	// Set the mode
	IF ctrl.nLS_Mode <> E_CRYO_LAKESHORE_MODE.MONITORING THEN
		Lakeshore.M_SetMode(ctrl.nLS_Mode);
	ELSE
		RETURN;	// Nothing to do
	END_IF
ELSE
	RETURN;	// Nothing to do
END_IF




CASE ctrl.nLS_Mode OF
	E_CRYO_LAKESHORE_MODE.MONITORING,
	E_CRYO_LAKESHORE_MODE.COOLING,
	E_CRYO_LAKESHORE_MODE.WARMUP,
	E_CRYO_LAKESHORE_MODE.COOLING_UPDATE,
	E_CRYO_LAKESHORE_MODE.WARMUP_UPDATE:
		Lakeshore.M_SetMode(E_CRYO_LAKESHORE_MODE.MONITORING);	// No action
		
	E_CRYO_LAKESHORE_MODE.SINGLE_SETUP:
		IF stat.nState = E_CRYO_CTRL_STATE.COLD THEN
			Lakeshore.M_SetParams(
				in_nPID_A_P			:= cfg.LS_W_PID_A_P, 
				in_nPID_A_I			:= cfg.LS_W_PID_A_I, 
				in_nPID_A_D			:= cfg.LS_W_PID_A_D, 
				in_nHeater_Range	:= cfg.LS_W_Heater_Range, 
				in_lrCtrlRamp		:= ctrl.lrLS_RAMP, 
				in_lrSetpoint_A		:= ctrl.lrLS_SETP);
		END_IF
	ELSE
		Lakeshore.M_SetMode(E_CRYO_LAKESHORE_MODE.MONITORING);	// No action
END_CASE
*)
END_METHOD

// Method to check status of the cryostat vacuum.
// TODO: The limits might depend on the temperature.
METHOD M_CheckVacuum
VAR_INPUT
END_VAR
//IF Pressure_Cryo.stat.bValid  THEN
//	IF Pressure_Cryo.stat.lrPressure < cfg.lrPress_GoodVac THEN
//		stat.bInVacuum	:= TRUE;
//		stat.bGoodVacuum:= TRUE;
//	ELSIF Pressure_Cryo.stat.lrPressure < cfg.lrPress_InVac THEN
//		stat.bInVacuum	:= TRUE;
//		stat.bGoodVacuum:= FALSE;
//	ELSE
//		stat.bInVacuum	:= FALSE;
//		stat.bGoodVacuum:= FALSE;
//	END_IF 
//ELSE
//	stat.bInVacuum	:= FALSE;
//	stat.bGoodVacuum:= FALSE;
//END_IF
END_METHOD

METHOD M_Configure
VAR_INPUT
END_VAR

IF NOT stat.bConfigured THEN
	

// This call just configures logs at the very start.
// Logging is done by explicit calls to M_LogInfo().
logs(in_sName := in_sName);

bPwr_VAG_PTA := TRUE;
bPwr_VAG_PTB := TRUE;
bPwr_VAG_PTC := TRUE;

	////////////////////
	// Coolant Valves//
	//////////////////
// Set pointers to Valves - MUST!!!
	ptrV[1]	:= ADR(TPC_A);
	ptrV[2]	:= ADR(TPC_B);
	
	
	// Set pointers to Valve Commands - MUST!!!
	ptrVC[1]	:= ADR(ctrl.cor_TPC_A);
	ptrVC[2]	:= ADR(ctrl.cor_TPC_B);
	
	
	// Set pointers to Enable Valves flags - MUST!!!
	ptrEV[1]	:= ADR(ctrl.bEnable_TPC_A);
	ptrEV[2]	:= ADR(ctrl.bEnable_TPC_B);









stat.bConfigured := TRUE;

END_IF 















//IF stat.bConfigured THEN
//	RETURN;
//ELSIF stat.nCycleCounter = 100 THEN
//	// Set pointers to system logs.
//	ptrLog[0] := ADR(syslog.s0);
//	ptrLog[1] := ADR(syslog.s1);
//	ptrLog[2] := ADR(syslog.s2);
//	ptrLog[3] := ADR(syslog.s3);
//	ptrLog[4] := ADR(syslog.s4);
//	ptrLog[5] := ADR(syslog.s5);
//	ptrLog[6] := ADR(syslog.s6);
//	ptrLog[7] := ADR(syslog.s7);
//	ptrLog[8] := ADR(syslog.s8);
//	ptrLog[9] := ADR(syslog.s9);
//ELSIF stat.nCycleCounter > 200 THEN
//	stat.bConfigured	:= TRUE;
//ELSE
//	RETURN;
//END_IF
END_METHOD

METHOD M_ExecuteControllers
VAR
END_VAR
VAR_INST
	trig_Turbo_ON:	R_TRIG;
	trig_Turbo_OFF:	F_TRIG;
END_VAR

met_tctrl(temperatures := met_temp);

met_heaters(tctrl := met_tctrl);

met_ccus();

// Evacuation is enabled, Check Venting valves and if they are open
// then Close them.
// Open PVV_P1 and Close PVV_P2 & PVV_P3
//IF met_evac.bEnable_met_evac THEN
//	IF met_venting.N2V_1.stat.bActON THEN
//		met_venting.in_bEnable_N2V_1 := FALSE;
//	END_IF
//	IF met_venting.N2V_2.stat.bActON THEN
//		met_venting.in_bEnable_N2V_2 := FALSE;
//	END_IF
	
//	met_cool_down.in_bEnable_PVV_P1:=	TRUE;
//	met_cool_down.in_bEnable_PVV_P2:=	FALSE;
//	met_cool_down.in_bEnable_PVV_P3:=	FALSE;
	
//	met_evac.stat.bInterlock := FALSE;
	
//END_IF


met_evac(in_Cryo_Stat := 						stat,
			interlocks:= 						interlocks);

//////////////////////////////////////////////
//             Venting
//////////////////////////////////////////////


met_venting(in_Cryo_Stat := 						stat,
			interlocks:= 						interlocks);

//////////////////////////////////////////////
//             Cool-Down
//////////////////////////////////////////////



met_cool_down(
	in_Cryo_Stat:=  							stat,
	in_lrLN2_TempK:= 							cfg.lrCoolDown_LN2_TempK,
	in_lrRadShld_TempK_TO_Start_PTCs:= 			cfg.lrRadShld_TempK_TO_Start_PTCs, 
	in_lrCoolDown_PreCond_Press:= 				cfg.lrCoolDown_PreCond_Press, 
	out_bCoolDownActive=> 						stat.bCoolDownActive, 
	all_cryo_temps:= 							met_temp, 
	all_heaters:= 								met_heaters, 
	all_t_ctrls:= 								met_tctrl, 
	all_t_votes:= 								met_voters, 
	interlocks:= 								interlocks);	





//////////////////////////////////////////////
//             Warmm_Up
//////////////////////////////////////////////

met_warm_up(
	in_Cryo_Stat:= 								stat, 
	in_lrWarmUp_Detectors_Ramp_1:= 				cfg.lrWarmUp_Detectors_Ramp_1, 
	in_lrWarmUp_Detectors_Ramp_Switch_Temp:=   	cfg.lrWarmUp_Detectors_Ramp_Switch_Temp, 
	in_lrWarmUp_Detectors_Ramp_2:=            	cfg.lrWarmUp_Detectors_Ramp_2,			
	in_lrWarmUp_EvacPermission_Temp:=         	cfg.lrWarmUp_EvacPermission_Temp,		
	in_lrWarmUp_VentingPermission_Temp:=      	cfg.lrWarmUp_VentingPermission_Temp,	
	in_lrWarmUp_Alarm_Temp:=                  	cfg.lrWarmUp_Alarm_Temp,				
	in_lrWarmUp_Alarm_PreCooling_Pressure:=   	cfg.lrWarmUp_Alarm_PreCooling_Pressure,
	out_bWarmUpActive=> 						stat.bWarmUpActive, 
	all_cryo_temps:= 							met_temp, 
	all_heaters:= 								met_heaters, 
	all_t_ctrls:= 								met_tctrl, 
	all_t_votes:= 								met_voters, 
	interlocks:= 								interlocks);



//////////////////////////////////////////////
//             Re_generation
//////////////////////////////////////////////


met_regeneration(
	in_Cryo_Stat:= 								stat, 
	in_lrRegeneration_Safe_Temp:= 				cfg.lrRegeneration_Safe_Temp, 
	in_lrRegeneration_Safe_Press:= 				cfg.lrRegeneration_Safe_Press, 
	in_lrTemp_Regeneration_SetPoint:= 			cfg.lrTemp_Regeneration_SetPoint, 
	in_lrTemp_Regeneration_Alarm:= 				cfg.lrTemp_Regeneration_Alarm_Temp, 
	in_lrTemp_Regeneration_Stop:= 				cfg.lrTemp_Regeneration_Stop, 
	in_tSorption_Pump_Cool_Down_TimeOut:= 		cfg.tSorption_Pump_Cool_Down_TimeOut, 
	out_bRegenerationActive=> 					stat.bRegenerationActive, 
	all_cryo_temps:= 							met_temp, 
	all_heaters:= 								met_heaters, 
	all_t_ctrls:= 								met_tctrl, 
	all_t_votes:=								met_voters, 
	interlocks:= 								interlocks);


//////////////////////////////////////////////
//             Anti-Fogging
//////////////////////////////////////////////


met_anti_fogging(
	//in_bEnable:= 								stat.bCoolDownActive, // Activate when Cool-down is active 
	in_Cryo_Stat:= 								stat, 
	in_lrAntiFog_Purging_DewPoint:= 			cfg.lrAntiFog_Purging_DewPoint, 
	in_lrAntiFog_Heating_DewPoint:= 			cfg.lrAntiFog_Heating_DewPoint, 
	in_lrAntiFog_DewPoint_Alarm:= 				cfg.lrAntiFog_DewPoint_Alarm, 
	out_bAntiFoggingActive=> 					stat.bAntiFoggingActive, 
	all_cryo_temps:= 							met_temp, 
	all_heaters:= 								met_heaters, 
	all_t_ctrls:= 								met_tctrl,   
	all_t_votes:=								met_voters,   
	interlocks:= 								interlocks);


//////////////////////////////////////////////
//             Coolant Valves
//////////////////////////////////////////////	

ctrl.cor_TPC_A(in_bEnable := ctrl.bEnable_TPC_A);	// Handling of PVV1 commands
ctrl.cor_TPC_B(in_bEnable := ctrl.bEnable_TPC_B);	// Handling of PVV2 commands

// Valve Control
TPC_A(
	in_bEnable			:= ctrl.cor_TPC_A.out_bEnable,
	in_nFeedback		:= E_CRYO_BIN_ACT_FEEDBACK.ON_ONLY);

TPC_B(
	in_bEnable			:= ctrl.cor_TPC_B.out_bEnable,
	in_nFeedback		:= E_CRYO_BIN_ACT_FEEDBACK.ON_ONLY);

// Reset valves

trig_Turbo_ON(CLK := stat.bTurboPumpsRunning);
trig_Turbo_OFF(CLK := stat.bTurboPumpsRunning);

IF trig_Turbo_ON.Q OR trig_Turbo_OFF.Q THEN
	TPC_A.M_Reset();
	TPC_B.M_Reset();
END_IF

// Actuate valves when turbo pumps are ON
ctrl.bEnable_TPC_A := stat.bTurboPumpsRunning;
ctrl.bEnable_TPC_B := stat.bTurboPumpsRunning;

	/////////////////////////////
	//// Time (NTP from ICS) /// 
	//////////////////////////

met_cry_time(in_diag_address:= , in_diag_destination_port:= , in_bDiagEnabled:= , in_nDefaultMode:= E_TIME_MODE.UTC_NTP);


	///////////////////////
	// xxxxxxxxxxxxxxxx //
	/////////////////////
	
	sim_regeneration();
END_METHOD

METHOD M_GetHighestTemperature
VAR_INPUT
END_VAR
VAR
	lrTempK:	LREAL	:= 0.0;	// The lowest possible temperature
	bValid:		BOOL	:= FALSE;
END_VAR
////
//// Get the warmest temperature among Mirror, Bench, FilterWheel and WarmUp
////

//// If there is at least one Valid reading, the result is valid.
//IF	Temp_Mirror.stat.bValid 	OR 
//	Temp_ColdBench.stat.bValid	OR 
//	Temp_FW.stat.bValid			OR 
//	Temp_WarmUp.stat.bValid			THEN
//	bValid	:= TRUE;
//END_IF


//// Get the highest temperature from Valid temperatures.
//// Take Mirror temperature first, if Valid.
//// If not Valid, try with WarmUp sensor.
//// If that doesn't work, take the Filter Wheel temperature.
//IF Temp_Mirror.stat.bValid THEN
//	IF Temp_Mirror.stat.lrTempK > lrTempK THEN
//		lrTempK	:= Temp_Mirror.stat.lrTempK;
//	END_IF
//ELSIF Temp_WarmUp.stat.bValid THEN
//	IF Temp_WarmUp.stat.lrTempK > lrTempK THEN
//		lrTempK	:= Temp_Mirror.stat.lrTempK;
//	END_IF
//ELSIF Temp_FW.stat.bValid THEN
//	IF Temp_FW.stat.lrTempK > lrTempK THEN
//		lrTempK	:= Temp_Mirror.stat.lrTempK;
//	END_IF
//END_IF


//// Update status
//stat.lrHighestTempK		:= lrTempK;
//stat.bHighestTempValid	:= bValid;
END_METHOD

METHOD M_GetLowestTemperature
VAR_INPUT
END_VAR
VAR
	lrTempK:	LREAL	:= 293.15;	// Room temperature 20 C
	bValid:		BOOL	:= FALSE;
END_VAR
////
//// Get the coldest temperature among Mirror, Bench, FilterWheel and WarmUp
////

//// If there is at least one Valid reading, the result is valid.
//IF	Temp_Mirror.stat.bValid 	OR 
//	Temp_ColdBench.stat.bValid	OR 
//	Temp_FW.stat.bValid			OR 
//	Temp_WarmUp.stat.bValid			THEN
//	bValid	:= TRUE;
//END_IF


//// Get the lowest temperature from Valid temperatures.
//IF Temp_Mirror.stat.bValid AND Temp_Mirror.stat.lrTempK < lrTempK THEN
//	lrTempK	:= Temp_Mirror.stat.lrTempK;
//END_IF

//IF Temp_ColdBench.stat.bValid AND Temp_ColdBench.stat.lrTempK < lrTempK THEN
//	lrTempK	:= Temp_ColdBench.stat.lrTempK;
//END_IF

//IF Temp_FW.stat.bValid AND Temp_FW.stat.lrTempK < lrTempK THEN
//	lrTempK	:= Temp_FW.stat.lrTempK;
//END_IF

//IF Temp_WarmUp.stat.bValid AND Temp_WarmUp.stat.lrTempK < lrTempK THEN
//	lrTempK	:= Temp_WarmUp.stat.lrTempK;
//END_IF

//// Update status
//stat.lrLowestTempK		:= lrTempK;
//stat.bLowestTempValid	:= bValid;

//// Get Temperature difference (DET -Lowest temperature) [K]
//IF stat.bLowestTempValid  AND  Temp_DET.stat.bValid  THEN
//	stat.bDiffTempValid	:= TRUE;
//	stat.lrDiffTempK	:= Temp_DET.stat.lrTempK - stat.lrLowestTempK;
//ELSE
//	stat.bDiffTempValid	:= FALSE;
//	stat.lrDiffTempK	:= -100;
//END_IF
END_METHOD

METHOD M_GetState
VAR_INPUT
END_VAR
VAR
	m_bIsCtrlOK           : BOOL;
    m_bIsWarm             : BOOL;
    m_bIsCold             : BOOL;
    m_bIsPartiallyCold    : BOOL;
    m_bIsInVacuum         : BOOL;
    m_bIsInPartialVacuum  : BOOL;
    m_bIsInGoodVacuum     : BOOL;
    m_bIsPressurized      : BOOL;

    m_nTmpState          : E_METIS_CRYO_CTRL_STATE;
    m_sStateDesc          : STRING;	

//    isCtrlOK: 			BOOL;
	
//    isWarm: 			BOOL;
//    isCold: 			BOOL;
//	isPartiallyCold: 	BOOL;
	
//    isInVacuum : 		BOOL;
//    isInPartialVacuum:	BOOL;
	
//	tempState : E_METIS_CRYO_CTRL_STATE;
END_VAR

m_bIsCtrlOK           := stat.bCtrlOK;
m_bIsWarm             := stat.bWarm;
m_bIsCold             := stat.bCold;
m_bIsPartiallyCold    := stat.bPartiallyCold;

m_bIsInVacuum         := stat.bInVacuum;
m_bIsInPartialVacuum  := stat.bPartialVacuum;
m_bIsInGoodVacuum     := stat.bInGoodVacuum;
m_bIsPressurized      := stat.bPressurized;


IF NOT m_bIsCtrlOK THEN
    m_nTmpState := E_METIS_CRYO_CTRL_STATE.ERROR;
    m_sStateDesc := 'Error: Controller is not OK';
	logs.M_LogInfo('');
	stat.bInitialized := FALSE;

ELSIF m_bIsWarm THEN
    IF m_bIsPressurized THEN
        m_nTmpState := E_METIS_CRYO_CTRL_STATE.WARM_PRESS;
        //m_sStateDesc := 'State: WarmPressurized';
		logs.M_LogInfo('System started in Warm-Pressurized state.');
		stat.bInitialized := TRUE;
    ELSIF m_bIsInVacuum THEN
        m_nTmpState := E_METIS_CRYO_CTRL_STATE.WARM_VACUUM;
        //m_sStateDesc := 'State: WarmVacuum';
		logs.M_LogInfo('System started in Warm-Vacuum state.');
		stat.bInitialized := TRUE;
    ELSIF m_bIsInPartialVacuum THEN
        m_nTmpState := E_METIS_CRYO_CTRL_STATE.PARTIAL_VACUUM;
        //m_sStateDesc := 'State: Partial Vacuum';
		logs.M_LogInfo('System started in Partial-Vacuum state');
		stat.bInitialized := TRUE;
    ELSE
        m_nTmpState := E_METIS_CRYO_CTRL_STATE.NONE;
        //m_sStateDesc := 'State Undefined: Warm with no pressure condition';
		logs.M_LogInfo('System started in undefined state: Warm with no pressure condition');
		stat.bInitialized := FALSE;
		ctrl.bEnable := FALSE;
    END_IF

ELSIF m_bIsCold THEN
	IF m_bIsInGoodVacuum THEN
    	m_nTmpState := E_METIS_CRYO_CTRL_STATE.COLD;
		logs.M_LogInfo('System started in Cold state');
		stat.bInitialized := TRUE;
	ELSE
		m_nTmpState := E_METIS_CRYO_CTRL_STATE.PARTIALLY_COLD;
		logs.M_LogInfo('System started in High Pressure & Low Temp state -> Start EVACUATION');
		stat.bInitialized := TRUE;
	END_IF

ELSIF m_bIsPartiallyCold THEN
    IF m_bIsInVacuum OR m_bIsInGoodVacuum THEN
        m_nTmpState := E_METIS_CRYO_CTRL_STATE.PARTIALLY_COLD;
       //m_sStateDesc := 'State: Partially Cold';
		logs.M_LogInfo('System started in Partially-Cold state.');
		stat.bInitialized := TRUE;
    ELSIF m_bIsPressurized THEN
        m_nTmpState := E_METIS_CRYO_CTRL_STATE.PARTIALLY_COLD;
        //m_sStateDesc := 'State: Partially Cold. Start EVACUATION';
		logs.M_LogInfo('System started in Partially-Cold state. Start EVACUATION');
		stat.bInitialized := TRUE;
    ELSE
        m_nTmpState := E_METIS_CRYO_CTRL_STATE.PARTIALLY_COLD;
        //m_sStateDesc := 'State: Partially Cold. Unknown pressure condition';
		logs.M_LogInfo('System started in Partially-Cold state with unknown pressure condition');
		stat.bInitialized := TRUE;
    END_IF

ELSE
    m_nTmpState := E_METIS_CRYO_CTRL_STATE.NONE;
    //m_sStateDesc := 'Critical Error: Undefined State -> Check System';
	logs.M_LogInfo('System started In Critical Error: Undefined State -> Check System');
	stat.bInitialized := FALSE;
	ctrl.bEnable := FALSE;
	logs.M_LogInfo('System Disabled...');
END_IF


stat.nState := m_nTmpState;
//stat.sState := m_sStateDesc;
M_SetStatus(stat.nState);

//logs.M_LogInfo(m_sStateDesc);



//isCtrlOK := stat.bCtrlOK;

//isWarm := stat.lrCryoTempK >= cfg.lrTemp_Cold;
//isCold := stat.lrCryoTempK <= cfg.lrTemp_Cold;
//isPartiallyCold := stat.bPartiallyCold;

//isInVacuum := stat.bInVacuum;
//isInPartialVacuum := stat.bPartialVacuum;



//IF NOT isCtrlOK THEN
//    tempState := E_METIS_CRYO_CTRL_STATE.ERROR;
//    stat.sState := 'Error: Controller is not OK';
//ELSE

//    IF isWarm AND stat.bPressurized THEN
//        tempState := E_METIS_CRYO_CTRL_STATE.WARM_PRESS;
//        stat.sState := 'State: Warm and Pressurized';
//    ELSIF isWarm AND isInVacuum THEN
//        tempState := E_METIS_CRYO_CTRL_STATE.WARM_VACUUM;
//        stat.sState := 'State: Warm and Vacuum';
//	ELSIF isWarm AND isInPartialVacuum THEN
//		tempState := E_METIS_CRYO_CTRL_STATE.PARTIAL_VACUUM;
//        stat.sState := 'State: Partial Vacuum';
	
//    ELSIF isCold AND stat.bInGoodVacuum THEN
//        tempState := E_METIS_CRYO_CTRL_STATE.COLD;
//        stat.sState := 'State: Cold';
		
//	ELSIF isPartiallyCold THEN
//		IF isInVacuum OR stat.bInGoodVacuum THEN
//			tempState := E_METIS_CRYO_CTRL_STATE.PARTIALLY_COLD;
//			stat.sState := 'State: Partially Cold';
//		ELSIF stat.bPressurized THEN
//			tempState := E_METIS_CRYO_CTRL_STATE.PARTIALLY_COLD;
//			stat.sState := 'State: Partially Cold. Start EVACUATION';
//		END_IF
//    ELSE        
//        tempState := E_METIS_CRYO_CTRL_STATE.NONE;
//        stat.sState := 'Critical Error: Undefined State -> Check System';
//    END_IF;
//END_IF;

//// 5.  Set the state.  This is done *once* at the end.
//stat.nState := tempState;
//M_SetStatus(stat.nState);
END_METHOD

METHOD M_HMI_Screen_Control : BOOL
VAR_INPUT
END_VAR
VAR_INST

    trigHMISwitch     : R_TRIG;  // Rising edge detector
	   bHMI_Enabled : BOOL;
END_VAR
	////////////////////
	//// HMI Screen /// 
	//////////////////
fuseHMI(in_sName:= 'Fuse - HMI Screen', in_bAutoOp:= TRUE, in_nTimeout:= );

bHMI_Enabled := fuseHMI.stat.stFuseStatus.bEnabled;

// Rising-edge detection on HMI switch
trigHMISwitch(CLK := bHMISwitch);


IF trigHMISwitch.Q THEN

    IF NOT bHMI_Enabled THEN

        fuseHMI.RPC_On();
    ELSE

        fuseHMI.RPC_Off();
    END_IF

END_IF
END_METHOD

METHOD PRIVATE M_ProcessHmi
// Vac Pumps

hmi_pump_tmp_a(
	inout_sPumpStatRef := met_evac.evac_branch_a.tp.stat,
	inout_sCmdOver := met_evac.evac_branch_a.cor_tp,
	inout_fbAlarmHandlerRef := met_evac.evac_branch_a.tp.fbAlarmHandler
	);

hmi_pump_pvp_a(
	inout_sPumpStatRef := met_evac.evac_branch_a.rp.stat,
	inout_sCmdOver := met_evac.evac_branch_a.cor_rp,
	inout_fbAlarmHandlerRef := met_evac.evac_branch_a.rp.fbAlarmHandler
	);

hmi_pump_tmp_b(
	inout_sPumpStatRef := met_evac.evac_branch_b.tp.stat,
	inout_sCmdOver := met_evac.evac_branch_b.cor_tp,
	inout_fbAlarmHandlerRef := met_evac.evac_branch_b.tp.fbAlarmHandler
	);

hmi_pump_pvp_b(
	inout_sPumpStatRef := met_evac.evac_branch_b.rp.stat,
	inout_sCmdOver := met_evac.evac_branch_b.cor_rp,
	inout_fbAlarmHandlerRef := met_evac.evac_branch_b.rp.fbAlarmHandler
	);

// Cryo Pressures
hmi_pressure_vote_vagf( inout_sPressureVoteStatRef := met_evac.VAGF.stat, inout_sCmdOver := met_evac.ctrl.por_VAGF , inout_fbAlarmHandlerRef := met_evac.VAGF.fbAlarmHandler);
hmi_pressure_vote_vagg( inout_sPressureVoteStatRef := met_evac.VAGG.stat, inout_sCmdOver := met_evac.ctrl.por_VAGG , inout_fbAlarmHandlerRef := met_evac.VAGG.fbAlarmHandler);

hmi_pressure_vote_vagg1( inout_sPressureVoteStatRef := met_evac.VAGG1.stat, inout_sCmdOver := met_evac.ctrl.por_VAGG1 , inout_fbAlarmHandlerRef := met_evac.VAGG1.fbAlarmHandler);
hmi_pressure_vote_vagg2( inout_sPressureVoteStatRef := met_evac.VAGG2.stat, inout_sCmdOver := met_evac.ctrl.por_VAGG2 , inout_fbAlarmHandlerRef := met_evac.VAGG2.fbAlarmHandler);

hmi_pressure_vote_vagf1( inout_sPressureVoteStatRef := met_evac.VAGF1.stat, inout_sCmdOver := met_evac.ctrl.por_VAGF1 , inout_fbAlarmHandlerRef := met_evac.VAGF1.fbAlarmHandler);
hmi_pressure_vote_vagf2( inout_sPressureVoteStatRef := met_evac.VAGF2.stat, inout_sCmdOver := met_evac.ctrl.por_VAGF2 , inout_fbAlarmHandlerRef := met_evac.VAGF2.fbAlarmHandler);

	
// Branch A
hmi_valve_pvv1_a( inout_sValveStatRef := met_evac.evac_branch_a.PVV1.stat,	inout_sCmdOver := met_evac.evac_branch_a.ctrl.cor_PVV1 , inout_fbAlarmHandlerRef := met_evac.evac_branch_a.PVV1.fbAlarmHandler);
hmi_valve_pvv2_a( inout_sValveStatRef := met_evac.evac_branch_a.PVV2.stat,	inout_sCmdOver := met_evac.evac_branch_a.ctrl.cor_PVV2 , inout_fbAlarmHandlerRef := met_evac.evac_branch_a.PVV2.fbAlarmHandler);
hmi_valve_pvv3_a( inout_sValveStatRef := met_evac.evac_branch_a.PVV3.stat,	inout_sCmdOver := met_evac.evac_branch_a.ctrl.cor_PVV3 , inout_fbAlarmHandlerRef := met_evac.evac_branch_a.PVV3.fbAlarmHandler);
hmi_valve_pvv4_a( inout_sValveStatRef := met_evac.evac_branch_a.PVV4.stat,	inout_sCmdOver := met_evac.evac_branch_a.ctrl.cor_PVV4 , inout_fbAlarmHandlerRef := met_evac.evac_branch_a.PVV4.fbAlarmHandler);
hmi_valve_GBV_a ( inout_sValveStatRef := met_evac.evac_branch_a.GBV.stat,	inout_sCmdOver := met_evac.evac_branch_a.ctrl.cor_GBV , inout_fbAlarmHandlerRef := met_evac.evac_branch_a.GBV.fbAlarmHandler);

hmi_pressure_vote_vag1_a( inout_sPressureVoteStatRef := met_evac.evac_branch_a.VAG1.stat, inout_sCmdOver := met_evac.evac_branch_a.ctrl.por_VAG1 , inout_fbAlarmHandlerRef := met_evac.evac_branch_a.VAG1.fbAlarmHandler);
hmi_pressure_vote_vag2_a( inout_sPressureVoteStatRef := met_evac.evac_branch_a.VAG2.stat, inout_sCmdOver := met_evac.evac_branch_a.ctrl.por_VAG2 , inout_fbAlarmHandlerRef := met_evac.evac_branch_a.VAG2.fbAlarmHandler);
hmi_pressure_vote_vag3_a( inout_sPressureVoteStatRef := met_evac.evac_branch_a.VAG3.stat, inout_sCmdOver := met_evac.evac_branch_a.ctrl.por_VAG3 , inout_fbAlarmHandlerRef := met_evac.evac_branch_a.VAG3.fbAlarmHandler);

// Branch B

hmi_valve_pvv1_b( inout_sValveStatRef := met_evac.evac_branch_b.PVV1.stat,	inout_sCmdOver := met_evac.evac_branch_b.ctrl.cor_PVV1 , inout_fbAlarmHandlerRef := met_evac.evac_branch_b.PVV1.fbAlarmHandler);
hmi_valve_pvv2_b( inout_sValveStatRef := met_evac.evac_branch_b.PVV2.stat,	inout_sCmdOver := met_evac.evac_branch_b.ctrl.cor_PVV2 , inout_fbAlarmHandlerRef := met_evac.evac_branch_b.PVV2.fbAlarmHandler);
hmi_valve_pvv3_b( inout_sValveStatRef := met_evac.evac_branch_b.PVV3.stat,	inout_sCmdOver := met_evac.evac_branch_b.ctrl.cor_PVV3 , inout_fbAlarmHandlerRef := met_evac.evac_branch_b.PVV3.fbAlarmHandler);
hmi_valve_pvv4_b( inout_sValveStatRef := met_evac.evac_branch_b.PVV4.stat,	inout_sCmdOver := met_evac.evac_branch_b.ctrl.cor_PVV4 , inout_fbAlarmHandlerRef := met_evac.evac_branch_b.PVV4.fbAlarmHandler);
hmi_valve_GBV_b ( inout_sValveStatRef := met_evac.evac_branch_b.GBV.stat,	inout_sCmdOver := met_evac.evac_branch_b.ctrl.cor_GBV , inout_fbAlarmHandlerRef := met_evac.evac_branch_b.GBV.fbAlarmHandler);

hmi_pressure_vote_vag1_b( inout_sPressureVoteStatRef := met_evac.evac_branch_b.VAG1.stat, inout_sCmdOver := met_evac.evac_branch_b.ctrl.por_VAG1 , inout_fbAlarmHandlerRef := met_evac.evac_branch_b.VAG1.fbAlarmHandler);
hmi_pressure_vote_vag2_b( inout_sPressureVoteStatRef := met_evac.evac_branch_b.VAG2.stat, inout_sCmdOver := met_evac.evac_branch_b.ctrl.por_VAG2 , inout_fbAlarmHandlerRef := met_evac.evac_branch_b.VAG2.fbAlarmHandler);
hmi_pressure_vote_vag3_b( inout_sPressureVoteStatRef := met_evac.evac_branch_b.VAG3.stat, inout_sCmdOver := met_evac.evac_branch_b.ctrl.por_VAG3 , inout_fbAlarmHandlerRef := met_evac.evac_branch_b.VAG3.fbAlarmHandler);


// PreCooling
hmi_valve_pvv_P1( inout_sValveStatRef := met_cool_down.PVV_P1.stat,	inout_sCmdOver := met_cool_down.ctrl.cor_PVV_P1 , inout_fbAlarmHandlerRef := met_cool_down.PVV_P1.fbAlarmHandler);
hmi_valve_pvv_P2( inout_sValveStatRef := met_cool_down.PVV_P2.stat,	inout_sCmdOver := met_cool_down.ctrl.cor_PVV_P2 , inout_fbAlarmHandlerRef := met_cool_down.PVV_P2.fbAlarmHandler);
hmi_valve_pvv_P3( inout_sValveStatRef := met_cool_down.PVV_P3.stat,	inout_sCmdOver := met_cool_down.ctrl.cor_PVV_P3 , inout_fbAlarmHandlerRef := met_cool_down.PVV_P3.fbAlarmHandler);

hmi_pressure_vote_vag_pca( inout_sPressureVoteStatRef := met_cool_down.VAG_PCA.stat, inout_sCmdOver := met_cool_down.ctrl.por_VAG_PCA , inout_fbAlarmHandlerRef := met_cool_down.VAG_PCA.fbAlarmHandler);
hmi_pressure_vote_vag_pcb( inout_sPressureVoteStatRef := met_cool_down.VAG_PCB.stat, inout_sCmdOver := met_cool_down.ctrl.por_VAG_PCB , inout_fbAlarmHandlerRef := met_cool_down.VAG_PCB.fbAlarmHandler);
hmi_pressure_vote_vag_p1 ( inout_sPressureVoteStatRef := met_cool_down.VAG_P1.stat,  inout_sCmdOver := met_cool_down.ctrl.por_VAG_P1 ,  inout_fbAlarmHandlerRef := met_cool_down.VAG_P1.fbAlarmHandler);


// Venting valves
hmi_valve_n2v1( inout_sValveStatRef := met_venting.N2V_1.stat,	inout_sCmdOver := met_venting.ctrl.cor_N2V_1 , inout_fbAlarmHandlerRef := met_venting.N2V_1.fbAlarmHandler);
hmi_valve_n2v2( inout_sValveStatRef := met_venting.N2V_2.stat,	inout_sCmdOver := met_venting.ctrl.cor_N2V_2 , inout_fbAlarmHandlerRef := met_venting.N2V_2.fbAlarmHandler);

// Water Cooling Valves
hmi_valve_tpc_A( inout_sValveStatRef := TPC_A.stat,	inout_sCmdOver :=ctrl.cor_TPC_A  , inout_fbAlarmHandlerRef := TPC_A.fbAlarmHandler);
hmi_valve_tpc_B( inout_sValveStatRef := TPC_B.stat,	inout_sCmdOver :=ctrl.cor_TPC_B  , inout_fbAlarmHandlerRef := TPC_B.fbAlarmHandler);

// LN2 Level Control Valves
hmi_valve_ln2_StifRingSeg     ( inout_sValveStatRef := met_cool_down.lc_ln2_level_ctrl[1].LN2_Valve.stat,	inout_sCmdOver :=  met_cool_down.lc_ln2_level_ctrl[1].cor_ln2_level_ctrl, inout_fbAlarmHandlerRef := met_cool_down.lc_ln2_level_ctrl[1].LN2_Valve.fbAlarmHandler); 		
hmi_valve_ln2_IntermediateSeg ( inout_sValveStatRef := met_cool_down.lc_ln2_level_ctrl[2].LN2_Valve.stat ,	inout_sCmdOver :=  met_cool_down.lc_ln2_level_ctrl[2].cor_ln2_level_ctrl, inout_fbAlarmHandlerRef := met_cool_down.lc_ln2_level_ctrl[2].LN2_Valve.fbAlarmHandler); 	
hmi_valve_ln2_BottomSeg       ( inout_sValveStatRef := met_cool_down.lc_ln2_level_ctrl[3].LN2_Valve.stat,	inout_sCmdOver :=  met_cool_down.lc_ln2_level_ctrl[3].cor_ln2_level_ctrl, inout_fbAlarmHandlerRef := met_cool_down.lc_ln2_level_ctrl[3].LN2_Valve.fbAlarmHandler); 		


// HPGs
hmi_pressure_vote_hpg ( inout_sPressureVoteStatRef := met_venting.HPG.stat,  inout_sCmdOver := met_venting.ctrl.por_HPG ,  inout_fbAlarmHandlerRef := met_venting.HPG.fbAlarmHandler);
hmi_pressure_vote_hpg1 ( inout_sPressureVoteStatRef := met_venting.HPG1.stat,  inout_sCmdOver := met_venting.ctrl.por_HPG1 ,  inout_fbAlarmHandlerRef := met_venting.HPG1.fbAlarmHandler);
hmi_pressure_vote_hpg2 ( inout_sPressureVoteStatRef := met_venting.HPG2.stat,  inout_sCmdOver := met_venting.ctrl.por_HPG2 ,  inout_fbAlarmHandlerRef := met_venting.HPG2.fbAlarmHandler);

// Coolers

	// Sleeves Pressures
	hmi_pressure_vote_vag_pta( inout_sPressureVoteStatRef := VAG_PTA.stat,  inout_sCmdOver := ctrl.por_VAG_PTA ,  inout_fbAlarmHandlerRef := VAG_PTA.fbAlarmHandler);
	hmi_pressure_vote_vag_ptb( inout_sPressureVoteStatRef := VAG_PTB.stat,  inout_sCmdOver := ctrl.por_VAG_PTB ,  inout_fbAlarmHandlerRef := VAG_PTB.fbAlarmHandler);
	hmi_pressure_vote_vag_ptc( inout_sPressureVoteStatRef := VAG_PTC.stat,  inout_sCmdOver := ctrl.por_VAG_PTC ,  inout_fbAlarmHandlerRef := VAG_PTC.fbAlarmHandler);

// LN2 Level Control Valves
hmi_valve_shav( inout_sValveStatRef := met_cool_down.lc_ln2_level_ctrl[1].LN2_Valve.stat, inout_sCmdOver := met_cool_down.lc_ln2_level_ctrl[1].cor_ln2_level_ctrl , inout_fbAlarmHandlerRef := met_cool_down.lc_ln2_level_ctrl[1].LN2_Valve.fbAlarmHandler);
hmi_valve_shbv( inout_sValveStatRef := met_cool_down.lc_ln2_level_ctrl[2].LN2_Valve.stat, inout_sCmdOver := met_cool_down.lc_ln2_level_ctrl[2].cor_ln2_level_ctrl , inout_fbAlarmHandlerRef := met_cool_down.lc_ln2_level_ctrl[2].LN2_Valve.fbAlarmHandler);
hmi_valve_shcv( inout_sValveStatRef := met_cool_down.lc_ln2_level_ctrl[3].LN2_Valve.stat, inout_sCmdOver := met_cool_down.lc_ln2_level_ctrl[3].cor_ln2_level_ctrl , inout_fbAlarmHandlerRef := met_cool_down.lc_ln2_level_ctrl[3].LN2_Valve.fbAlarmHandler);
END_METHOD

METHOD M_ReadSensors
VAR_INPUT
END_VAR


sensor_VAG_PTA(in_sName:= 'VAG_PTA', in_nType:= E_CRYO_SENSOR_TYPE_PRESS.PKR_360, in_lrBitsPerVolt:= , in_nSampleTime:= 100);
sensor_VAG_PTB(in_sName:= 'VAG_PTB', in_nType:= E_CRYO_SENSOR_TYPE_PRESS.PKR_360, in_lrBitsPerVolt:= , in_nSampleTime:= 100);
sensor_VAG_PTC(in_sName:= 'VAG_PTC', in_nType:= E_CRYO_SENSOR_TYPE_PRESS.PKR_360, in_lrBitsPerVolt:= , in_nSampleTime:= 100);

ctrl.por_VAG_PTA(in_bEnable := ctrl.bSim_Press_VAG_PTA);	// Simulation flag override
VAG_PTA(
	in_sName:= 'VAG_PTA', 
	in_bSimulation:= ctrl.por_VAG_PTA.out_bEnable, 
	in_nNumSensor:= 1, 
	in_nVoteMethod:= , 
	in_pSensor1:= ADR(sensor_VAG_PTA), 
	in_pSensor2:= , 
	in_pSensor3:= , 
	in_pSensor4:= , 
	in_pSensor5:= );
	
ctrl.por_VAG_PTB(in_bEnable := ctrl.bSim_Press_VAG_PTB);	// Simulation flag override
VAG_PTB(
	in_sName:= 'VAG_PTB', 
	in_bSimulation:= ctrl.por_VAG_PTB.out_bEnable, 
	in_nNumSensor:= 1, 
	in_nVoteMethod:= , 
	in_pSensor1:= ADR(sensor_VAG_PTB), 
	in_pSensor2:= , 
	in_pSensor3:= , 
	in_pSensor4:= , 
	in_pSensor5:= );
	
ctrl.por_VAG_PTC(in_bEnable := ctrl.bSim_Press_VAG_PTC);	// Simulation flag override
VAG_PTC(
	in_sName:= 'VAG_PTC', 
	in_bSimulation:= ctrl.por_VAG_PTC.out_bEnable, 
	in_nNumSensor:= 1, 
	in_nVoteMethod:= , 
	in_pSensor1:= ADR(sensor_VAG_PTC), 
	in_pSensor2:= , 
	in_pSensor3:= , 
	in_pSensor4:= , 
	in_pSensor5:= );

	///////////////////////
	// Ambient Pressure //
	/////////////////////

sensor_AMB_PRESS(in_sName:= 'Ambient Pressure' , in_lrBitsPerVolt:= , in_nSampleTime:= );	

stat.lrAmbientPressure := sensor_AMB_PRESS.stat.lrPressure;


// Read temperatures
met_temp();

// Update the voters
met_voters(met_temp := met_temp);

// Read relative humidities
met_rh(met_temp := met_temp);
END_METHOD

METHOD M_SafetyCheck
VAR_INPUT
END_VAR
////
//// Repressurization safety
////
//IF	NOT ctrl.bEnable_Evac AND
//	(stat.nState = E_CRYO_CTRL_STATE.WARM_PRESS 		OR 
//	 stat.nState = E_CRYO_CTRL_STATE.REPRESSURIZING 	OR 
//	 stat.nState = E_CRYO_CTRL_STATE.WARM_VACUUM) 		THEN
//	ctrl.bSafe_Repress	:= TRUE;
//ELSE
//	ctrl.bSafe_Repress	:= FALSE;
//	ctrl.bEnable_RepressSys:= FALSE;
//END_IF


M_CheckDetectorsSafety();
END_METHOD

METHOD PRIVATE M_SetError
VAR_INPUT
    nCode     : UDINT;
    sMessage  : STRING;
END_VAR


stat.Error.nCode := nCode;
stat.Error.sMessage := sMessage;
stat.bError := TRUE;
stat.nState := E_METIS_CRYO_CTRL_STATE.ERROR;
END_METHOD

METHOD M_SetStatus
VAR_INPUT
	nState:	E_METIS_CRYO_CTRL_STATE;
END_VAR
// TODO: Re-visit the following implementation of estimating nState when no sequence is running. 
//IF NOT stat.bBusy THEN
//	M_GetState();
//END_IF 




CASE nState OF
	
	E_METIS_CRYO_CTRL_STATE.NONE:
	
	stat.bDone	:= TRUE;
	stat.bBusy	:= FALSE;
	stat.bError	:= FALSE;
	stat.bActive:= FALSE;
	stat.sState	:= 'OFF';
	IF stat.bEvacuationActive THEN
		stat.bDone	:= FALSE;
		stat.bBusy	:= TRUE;
		stat.bError	:= FALSE;
		stat.bActive:= TRUE;
		stat.sState	:= 'EVACUATING...';
	END_IF
	
	E_METIS_CRYO_CTRL_STATE.WARM_PRESS:
	
	stat.bDone	:= TRUE;
	stat.bBusy	:= FALSE;
	stat.bError	:= FALSE;
	stat.bActive:= TRUE;
	stat.sState	:= 'WARM  -  PRESSURIZED';
	
	E_METIS_CRYO_CTRL_STATE.PARTIAL_VACUUM:
	
	stat.bDone	:= TRUE;
	stat.bBusy	:= FALSE;
	stat.bError	:= FALSE;
	stat.bActive:= TRUE;
	stat.sState	:= 'PARTIAL VACUUM';

	IF stat.bEvacuationActive THEN
		stat.bDone	:= FALSE;
		stat.bBusy	:= TRUE;
		stat.bError	:= FALSE;
		stat.bActive:= TRUE;
		stat.sState	:= 'EVACUATING...';
	END_IF
	
	E_METIS_CRYO_CTRL_STATE.WARM_VACUUM:
	
	stat.bDone	:= TRUE;
	stat.bBusy	:= FALSE;
	stat.bError	:= FALSE;
	stat.bActive:= TRUE;
	stat.sState	:= 'WARM  -  VACUUM';
	

	E_METIS_CRYO_CTRL_STATE.COOLING_DOWN:
	
	stat.bDone	:= FALSE;
	stat.bBusy	:= TRUE;
	stat.bError	:= FALSE;
	stat.bActive:= TRUE;
	stat.sState	:= 'COOLING DOWN...';
	
	E_METIS_CRYO_CTRL_STATE.PARTIALLY_COLD:
	
	stat.bDone	:= TRUE;
	stat.bBusy	:= FALSE;
	stat.bError	:= FALSE;
	stat.bActive:= TRUE;
	stat.sState	:= 'PARTIALLY COLD';

	E_METIS_CRYO_CTRL_STATE.COLD:
	
	stat.bDone	:= TRUE;
	stat.bBusy	:= FALSE;
	stat.bError	:= FALSE;
	stat.bActive:= TRUE;
	stat.sState	:= 'COLD';

	E_METIS_CRYO_CTRL_STATE.WARMING_UP:
	
	stat.bDone	:= FALSE;
	stat.bBusy	:= TRUE;
	stat.bError	:= FALSE;
	stat.bActive:= TRUE;
	IF stat.lrCryoTempK >= cfg.lrTemp_Warm	THEN
		stat.sState	:= 'WARM';
	ELSE
		stat.sState	:= 'WARMING UP...';
	END_IF

	E_METIS_CRYO_CTRL_STATE.VENTING:
	
	stat.bDone	:= FALSE;
	stat.bBusy	:= TRUE;
	stat.bError	:= FALSE;
	stat.bActive:= TRUE;
	stat.sState	:= 'VENTING...';
	
	E_METIS_CRYO_CTRL_STATE.ERROR:
	
	stat.bDone	:= TRUE;
	stat.bBusy	:= FALSE;
	stat.bError	:= TRUE;
	stat.bActive:= FALSE;
	stat.sState	:= 'ERROR';

END_CASE
END_METHOD

METHOD M_StateMachine
VAR_INPUT
END_VAR
VAR_INST
	bStarted:			BOOL := FALSE;
	Start_Timer:		TON;
	tStart_TimeOut:		TIME := T#30S;
		
	
	Init_Timer:			TON;
	tInit_TimeOut:		TIME := cfg.tInitTimeOut;
	bLogToggle:			BOOL := FALSE;
END_VAR
////////////////
// State Machine
////////////////
CASE stat.nState OF
	
	/////////////////////////////////
	E_METIS_CRYO_CTRL_STATE.NONE:
	/////////////////////////////////

		M_Activity_None();

	/////////////////////////////////
	E_METIS_CRYO_CTRL_STATE.WARM_PRESS:
	/////////////////////////////////

		M_Activity_Warm_Press_State();
	
	/////////////////////////////////
	E_METIS_CRYO_CTRL_STATE.PARTIAL_VACUUM:
	/////////////////////////////////
	
		M_Activity_Partial_Vacuum_State();
	
	/////////////////////////////////
	E_METIS_CRYO_CTRL_STATE.VENTING:
	/////////////////////////////////
	
		M_Activity_Venting();
	
	//////////////////////////////////////////
	E_METIS_CRYO_CTRL_STATE.WARM_VACUUM:
	//////////////////////////////////////////

		M_Activity_Warm_Vacuum_State();
	
	/////////////////////////////////
	E_METIS_CRYO_CTRL_STATE.COOLING_DOWN:
	/////////////////////////////////
	
		M_Activity_Cooling_Down_State();
	
	/////////////////////////////////////////
	E_METIS_CRYO_CTRL_STATE.PARTIALLY_COLD:
	////////////////////////////////////////
	
		M_Activity_Partially_Cold_State(); 
	
	///////////////////////////////////////////
	E_METIS_CRYO_CTRL_STATE.COLD:
	///////////////////////////////////////////
	
		M_Activity_Cold_State();
	
	/////////////////////////////////
	E_METIS_CRYO_CTRL_STATE.WARMING_UP:
	/////////////////////////////////
	
		M_Activity_Warm_Up_State();
	
	/////////////////////////////////
	E_METIS_CRYO_CTRL_STATE.ERROR:
	/////////////////////////////////

		M_Activity_Error_State();

END_CASE



//////////////////
//// State Machine
//////////////////
//CASE stat.nState OF
	
//	/////////////////////////////////
//	E_METIS_CRYO_CTRL_STATE.NONE:
//	/////////////////////////////////
//		// This is the state on power-up.
//		IF NOT bStarted THEN
//			bStarted := TRUE;	
//			Start_Timer(IN := TRUE, PT := tStart_TimeOut);
//			RETURN;
//		END_IF
		
//		IF Start_Timer.Q THEN	
//			M_GetState();
//			Start_Timer(IN := FALSE);
//			RETURN;
//		ELSE
//			RETURN;
//		END_IF
		
		
//		IF NOT (stat.nState = E_METIS_CRYO_CTRL_STATE.WARM_PRESS) THEN
//			M_Activity_Stabilize_Cryostat_Conditions();
//			stat.nState := E_METIS_CRYO_CTRL_STATE.NONE;
//			RETURN;
//		END_IF
		
		
//		// Determine the initial state based on the command and actuator state.
//		IF ctrl.bEnable THEN
//			IF NOT bLogToggle THEN
//				logs.M_LogInfo('System enabled...');
//				logs.M_LogInfo('Initializing controller...');
//				bLogToggle := TRUE;
//			END_IF
//			Init_Timer(IN := TRUE, PT := tInit_TimeOut);
//			IF	Init_Timer.Q THEN
//				M_GetState();
//			ELSE
				
//				stat.sState := 'Initializing Controller...';
//				stat.bActive := TRUE;
//				IF trgSystemDisable.Q THEN
//					stat.sState := 'Initialization Aborted';
//					stat.bActive := FALSE;
//					ctrl.nCommand		:= E_METIS_CRYO_CTRL_CMD.NONE;
//				END_IF
//				RETURN;
//			END_IF
			
//		ELSE
//			stat.bActive := FALSE;
//			stat.sState := 'Inactive: Enable When Ready';
//			RETURN;
//		END_IF
		
//		RETURN;
	

//	/////////////////////////////////
//	E_METIS_CRYO_CTRL_STATE.WARM_PRESS:
//	/////////////////////////////////
//	//
//	ctrl.bSafe_Evac 		:= TRUE;
//	ctrl.bSafe_Cool_Down 	:= FALSE;
//	ctrl.bSafe_Warm_Up		:= FALSE;
//	ctrl.bSafe_Regeneration := FALSE;
//	ctrl.bEnable_Venting 	:= FALSE;


//	IF	ctrl.bExecute	THEN
//		ctrl.bExecute		:= FALSE;
//		stat.nLastCommand	:= ctrl.nCommand;
//		ctrl.nCommand		:= E_METIS_CRYO_CTRL_CMD.NONE;
//		IF stat.nLastCommand = E_METIS_CRYO_CTRL_CMD.NONE THEN
//			logs.M_LogInfo('Cryo Controller Disables by operator');
//			stat.nState	:= E_METIS_CRYO_CTRL_STATE.NONE;
//			ctrl.bEnable := FALSE;
//			stat.bInitialized := FALSE;
//			Init_Timer(IN := FALSE);
//		END_IF
//	ELSIF stat.bPartialVacuum THEN
//		// Evacuation is not part of the State Machine.
//		// Once the pressure is below ambient , we switch to Partial Vacuum.
//		stat.nState := E_METIS_CRYO_CTRL_STATE.PARTIAL_VACUUM;
//		logs.M_LogInfo('Partial Vacuum Achieved');
//	END_IF
//	M_SetStatus(stat.nState);	
//	RETURN;
	
//	/////////////////////////////////
//	E_METIS_CRYO_CTRL_STATE.PARTIAL_VACUUM:
//	/////////////////////////////////
	
//	ctrl.bSafe_Evac 		:= TRUE;
//	ctrl.bSafe_Cool_Down 	:= FALSE;
//	ctrl.bSafe_Warm_Up		:= FALSE;
//	ctrl.bSafe_Regeneration := FALSE;
//	ctrl.bSafe_Venting 		:= TRUE;


//	IF	ctrl.bExecute	THEN
//		ctrl.bExecute		:= FALSE;
//		stat.nLastCommand	:= ctrl.nCommand;
//		ctrl.nCommand		:= E_METIS_CRYO_CTRL_CMD.NONE;
//		IF stat.nLastCommand = E_METIS_CRYO_CTRL_CMD.VENT THEN
//			logs.M_LogInfo('VENTING initiated by operator');
//			stat.nState	:= E_METIS_CRYO_CTRL_STATE.VENTING;
//		END_IF
//	ELSIF stat.bInVacuum OR stat.bInGoodVacuum THEN
//		stat.nState := E_METIS_CRYO_CTRL_STATE.WARM_VACUUM;
//		logs.M_LogInfo('Vacuum Achieved');
//	END_IF
//	M_SetStatus(stat.nState);	
//	RETURN;
	
//	/////////////////////////////////
//	E_METIS_CRYO_CTRL_STATE.VENTING:
//	/////////////////////////////////
//	//
//	ctrl.bSafe_Cool_Down 	:= FALSE;
//	ctrl.bSafe_Warm_Up 		:= FALSE;
//	ctrl.bSafe_Evac 		:= FALSE;
//	ctrl.bSafe_Regeneration := FALSE;


//	IF	stat.bVentingFinishedSuccessfully  THEN
		
//		ctrl.bEnable_Venting := FALSE;

//		logs.M_LogInfo('VENTING Finished');
//		stat.nState	:= E_METIS_CRYO_CTRL_STATE.WARM_PRESS;
//		logs.M_LogInfo('State is Warm-Pressurized');
//	ELSIF trgVentingOff.Q THEN
//		// Re-pressurization has been interrupted.
//		logs.M_LogInfo('VENTING interrupted by operator...');

//		IF stat.bPressurized THEN
//			stat.nState := E_METIS_CRYO_CTRL_STATE.WARM_PRESS;
//			logs.M_LogInfo('State is Warm-Pressurized');
//		ELSIF stat.bPartialVacuum THEN
//			stat.nState := E_METIS_CRYO_CTRL_STATE.PARTIAL_VACUUM;
//			logs.M_LogInfo('State is Partial Vacuum');
//		ELSIF stat.bInVacuum OR stat.bInGoodVacuum THEN
//			stat.nState := E_METIS_CRYO_CTRL_STATE.WARM_VACUUM;
//			logs.M_LogInfo('State is Warm Vacuum'); 
//		END_IF
		
//	END_IF
//	M_SetStatus(stat.nState);	
//	RETURN;
	
//	//////////////////////////////////////////
//	E_METIS_CRYO_CTRL_STATE.WARM_VACUUM:
//	//////////////////////////////////////////
//	//
//	ctrl.bSafe_Evac			:= TRUE;
//	ctrl.bSafe_Venting		:= TRUE;
//	ctrl.bSafe_Cool_Down	:= TRUE;
//	ctrl.bSafe_Regeneration := TRUE;

//	IF	ctrl.bExecute	THEN
//		ctrl.bExecute		:= FALSE;
//		stat.nLastCommand	:= ctrl.nCommand;
//		ctrl.nCommand		:= E_METIS_CRYO_CTRL_CMD.NONE;
//		IF stat.nLastCommand = E_METIS_CRYO_CTRL_CMD.COOL	THEN	
//			logs.M_LogInfo('Cool-Down initiated by operator');
//			stat.nState	:= E_METIS_CRYO_CTRL_STATE.COOLING_DOWN;
//		ELSIF stat.nLastCommand = E_METIS_CRYO_CTRL_CMD.VENT	THEN
//			logs.M_LogInfo('VENTING initiated by operator');
//			stat.nState	:= E_METIS_CRYO_CTRL_STATE.VENTING;
//		END_IF
//	END_IF
//	M_SetStatus(stat.nState);	
//	RETURN;
	
	
//	/////////////////////////////////
//	E_METIS_CRYO_CTRL_STATE.COOLING_DOWN:
//	/////////////////////////////////
//	//
//	ctrl.bSafe_Evac 			:= TRUE;
//	ctrl.bSafe_Cool_Down 		:= TRUE;
//	ctrl.bSafe_Warm_Up 			:= FALSE;
//	ctrl.bSafe_Regeneration 	:= FALSE;
//	ctrl.bSafe_Anti_Fogging		:= TRUE;
//	ctrl.bSafe_Venting 			:= FALSE;
//	ctrl.bEnable_Venting		:= FALSE;
//	stat.bPermitEvacuationStop 	:= FALSE;
	
//	IF NOT stat.bCoolDownActive THEN
//		ctrl.bEnable_Cool_Down := FALSE;
//	END_IF
//	IF stat.bOP THEN
//		logs.M_LogInfo('Cool-Down complete. State is Cold.');
//		stat.nState	:= E_METIS_CRYO_CTRL_STATE.COLD;
//	ELSIF trgCoolOFF.Q THEN
//		// Cooling has been interrupted.
//		logs.M_LogInfo('Cooling interrupted by operator OR error...');
		
//		IF stat.bOP THEN
//			logs.M_LogInfo('Cool-Down complete. State is Cold and ready for operations.');
//			stat.nState	:= E_METIS_CRYO_CTRL_STATE.COLD;
//		ELSIF stat.bPartiallyCold THEN 
//			logs.M_LogInfo('State is Partially Cold.');
//			stat.nState	:= E_METIS_CRYO_CTRL_STATE.PARTIALLY_COLD;
//		ELSIF stat.bWarm THEN
//			logs.M_LogInfo('State is Warm Vacuum');
//			stat.nState	:= E_METIS_CRYO_CTRL_STATE.WARM_VACUUM;
//		END_IF
		
//	END_IF
//	M_SetStatus(stat.nState);	
//	RETURN;

//	/////////////////////////////////////////
//	E_METIS_CRYO_CTRL_STATE.PARTIALLY_COLD:
//	////////////////////////////////////////
	
//	ctrl.bSafe_Evac 			:= TRUE;
//	ctrl.bSafe_Cool_Down 		:= TRUE;
//	ctrl.bSafe_Warm_Up 			:= TRUE;
//	ctrl.bSafe_Regeneration 	:= FALSE;
//	ctrl.bSafe_Anti_Fogging		:= TRUE;
//	ctrl.bSafe_Venting 			:= FALSE;
//	ctrl.bEnable_Venting		:= FALSE;
//	stat.bPermitEvacuationStop 	:= FALSE;
	
//	IF	ctrl.bExecute	THEN
//		ctrl.bExecute		:= FALSE;
//		stat.nLastCommand	:= ctrl.nCommand;
//		ctrl.nCommand		:= E_METIS_CRYO_CTRL_CMD.NONE;
//		IF stat.nLastCommand = E_METIS_CRYO_CTRL_CMD.COOL	THEN	
//			logs.M_LogInfo('Cool-Down initiated by operator');
//			stat.nState	:= E_METIS_CRYO_CTRL_STATE.COOLING_DOWN;
//		ELSIF stat.nLastCommand = E_METIS_CRYO_CTRL_CMD.WARM_UP	THEN
//			logs.M_LogInfo('Warm-Up initiated by operator');
//			stat.nState	:= E_METIS_CRYO_CTRL_STATE.WARMING_UP;
//		END_IF
//	ELSE
//		M_Activity_Stabilize_Cryostat_Conditions();
//		stat.nState	:= E_METIS_CRYO_CTRL_STATE.PARTIALLY_COLD;
//	END_IF
	
//	M_SetStatus(stat.nState);	
//	RETURN;
	
//	///////////////////////////////////////////
//	E_METIS_CRYO_CTRL_STATE.COLD:
//	///////////////////////////////////////////
//	//
//	ctrl.bSafe_Evac 			:= TRUE;
//	ctrl.bSafe_Cool_Down 		:= FALSE;
//	ctrl.bSafe_Warm_Up 			:= FALSE;
//	ctrl.bSafe_Regeneration 	:= FALSE;
//	ctrl.bSafe_Venting 			:= FALSE;
//	ctrl.bEnable_Venting		:= FALSE;
//	ctrl.bSafe_Anti_Fogging		:= TRUE;
//	stat.bPermitEvacuationStop 	:= TRUE;
	
//	//
//	// Only WARM_UP command is allowed in state COLD.

//	IF	ctrl.bExecute	THEN
//		ctrl.bExecute		:= FALSE;
//		stat.nLastCommand	:= ctrl.nCommand;
//		ctrl.nCommand		:= E_METIS_CRYO_CTRL_CMD.NONE;
//		IF stat.nLastCommand = E_METIS_CRYO_CTRL_CMD.WARM_UP	THEN
			
//			ctrl.bSafe_Warm_Up := TRUE;
//			IF NOT ctrl.bEnable_Evac THEN 
//				ctrl.bEnable_Evac  := TRUE;
//			END_IF
			
//			logs.M_LogInfo('Warm-Up initiated by operator');
//			stat.nState	:= E_METIS_CRYO_CTRL_STATE.WARMING_UP;
//		END_IF
//	ELSE
//		met_cool_down.M_Activity_Cold_State();
//		stat.nState	:= E_METIS_CRYO_CTRL_STATE.COLD;
//	END_IF
//	M_SetStatus(stat.nState);	
//	RETURN;
	
//	/////////////////////////////////
//	E_METIS_CRYO_CTRL_STATE.WARMING_UP:
//	/////////////////////////////////
//	//
//	ctrl.bSafe_Evac 			:= TRUE;
//	ctrl.bSafe_Cool_Down 		:= FALSE;
//	ctrl.bSafe_Warm_Up 			:= TRUE;
//	ctrl.bSafe_Regeneration 	:= FALSE;
//	ctrl.bSafe_Venting 			:= FALSE;
//	ctrl.bEnable_Venting		:= FALSE;
//	ctrl.bSafe_Anti_Fogging		:= FALSE;
//	stat.bPermitEvacuationStop 	:= FALSE;
	
//	ctrl.bSafe_Cool_Down 		:= FALSE;
//	ctrl.bSafe_Regeneration 	:= FALSE;
//	ctrl.bSafe_Venting 			:= FALSE;
//	ctrl.bEnable_Venting		:= FALSE;

//	IF trgWarmupOff.Q THEN
//		ctrl.bEnable_Warm_Up	:= FALSE;
//		IF	stat.bWarm THEN
//				logs.M_LogInfo('Warming up complete. State is Warm-Vaccum');
//				stat.nState := E_METIS_CRYO_CTRL_STATE.WARM_VACUUM;
//		ELSIF stat.bPartiallyCold THEN
//				logs.M_LogInfo('Warming up complete. State is Partially-Cold');
//				stat.nState := E_METIS_CRYO_CTRL_STATE.PARTIALLY_COLD;
//		ELSIF stat.bOP THEN
//				logs.M_LogInfo('Warming up complete. State is Cold');
//				stat.nState := E_METIS_CRYO_CTRL_STATE.COLD;
//		END_IF		
//	END_IF
//	M_SetStatus(stat.nState);	
//	RETURN;
	
//	/////////////////////////////////
//	E_METIS_CRYO_CTRL_STATE.ERROR:
//	/////////////////////////////////
//	//
//	// RESET the controller in order to try to clear error
//	IF ctrl.bReset THEN
//		ctrl.bReset	:= FALSE;	// Clear RESET flag
//		// Goto NONE state
//		stat.nState	:= E_METIS_CRYO_CTRL_STATE.NONE;
//		stat.bInitialized := FALSE;
//		M_SetStatus(stat.nState);	
//	ELSIF NOT stat.bError  THEN
//		// Goto NONE state
//		stat.nState	:= E_METIS_CRYO_CTRL_STATE.NONE;
//		stat.bInitialized := FALSE;
//		M_SetStatus(stat.nState);	
//	END_IF
//	RETURN;

//END_CASE
END_METHOD

METHOD M_SysLog
VAR_INPUT
	str:	STRING(80);
END_VAR
VAR
	i:	INT;
END_VAR
//nLogPos	:= nLogPos + 1;
//IF nLogPos > 9 THEN
//	FOR i := 1 TO 9 DO
//		// Shift last 9 readings
//		ptrLog[i-1]^ := ptrLog[i]^;
//	END_FOR
//	nLogPos	:= 9;
//END_IF

//ptrLog[nLogPos]^ := str;
END_METHOD

METHOD M_UpdatePressureStates : BOOL
VAR_INPUT
END_VAR
VAR
	bInGoodVacuuumCond:	BOOL;
	bInVacuumCond:		BOOL;
	bPressurizedCond:	BOOL;
END_VAR
stat.lrVAGF := met_evac.VAGF.stat.lrPressure;
stat.lrVAGG := met_evac.VAGG.stat.lrPressure;
stat.lrHPG  := met_venting.HPG.stat.lrPressure;

bPressurizedCond 	:= (stat.lrHPG  > cfg.lrPress_Atm); // OR (stat.lrVAGF > cfg.lrPress_Atm) OR (stat.lrVAGG > cfg.lrPress_Atm);
bInVacuumCond    	:= (stat.lrVAGF < cfg.lrPress_InVac) OR (stat.lrVAGG < cfg.lrPress_InVac);
bInGoodVacuuumCond	:= (stat.lrVAGF < cfg.lrPress_GoodVac) OR (stat.lrVAGG < cfg.lrPress_GoodVac);


(* Edge detection: Rising edge when entering vacuum or becoming pressurized *)
trgPressurized(CLK := bPressurizedCond);
trgInVaccum(CLK := bInVacuumCond);
trgInGoodVaccum(CLK := bInGoodVacuuumCond);


(* Set flags based on conditions or trigger events *)

stat.bPressurized 	:= bPressurizedCond OR trgPressurized.Q;
stat.bInVacuum 		:= bInVacuumCond OR trgInVaccum.Q;
stat.bInGoodVacuum 	:= bInGoodVacuuumCond OR trgInGoodVaccum.Q;

(* Determine partial vacuum state when neither vacuum nor pressurized is active *)
stat.bPartialVacuum := (stat.lrHPG  < cfg.lrPress_Atm) AND (NOT (stat.bInGoodVacuum OR stat.bInVacuum)); //NOT stat.bInVacuum AND NOT stat.bPressurized;
END_METHOD

METHOD M_UpdateStatus
VAR

	
	bColdCond:			BOOL;
	bWarmCond:			BOOL;
END_VAR

// Routine Active Status

stat.bEvacuationActive 		:= met_evac.out_bEvacuationActive;
stat.bVentingActive 		:= met_venting.out_bVentingActive;
stat.bCoolDownActive 		:= met_cool_down.out_bCoolDownActive;
stat.bWarmUpActive 			:= met_warm_up.out_bWarmUpActive;
stat.bRegenerationActive 	:= met_regeneration.out_bRegenerationActive;
stat.bAntiFoggingActive 	:= met_anti_fogging.out_bAntiFoggingActive;
stat.bPowerOutageActive 	:= met_power_outage.out_bPowerOutageActive;
stat.bStopPowerOutageActive := met_stop_power_outage.out_bStopPowerOutageActive;


		 ////////////////////////////////
		//// Safe To Disable System ////
	   ////////////////////////////////
	   
IF stat.nState = E_METIS_CRYO_CTRL_STATE.NONE 
	OR stat.nState = E_METIS_CRYO_CTRL_STATE.WARM_PRESS THEN
 
	stat.bSafeToDisableSystem := TRUE;
ELSE
	stat.bSafeToDisableSystem := FALSE;
END_IF

		 ///////////////////////////////////////
		//// Permission to stop Evacuation ////
	   ///////////////////////////////////////

	
stat.bPermitEvacuationStop := met_cool_down.M_PermitEvacuationStop() OR 
								met_warm_up.M_PermitEvacuationStop() OR
								met_regeneration.M_PermitEvacuationStop(); 
 
		 ///////////////////////////////////////
		//// Statuses of critical devices ////
	   ///////////////////////////////////////

stat.bVentingValvesAreClosed := met_venting.M_AreVentingValvesClosed();  
stat.bPumpsAreRunning := met_evac.M_AreAnyPumpsRunning();	
stat.bRoughingPumpsAreRunning := met_evac.M_AreRoughingPumpRunning();
stat.bTurboPumpsRunning	:= met_evac.M_AreTurboPumpsRunning();


// 
stat.bWarmUpHeatersActive := met_warm_up.M_AreWarmUpHeaterActive();				




		 ///////////////////////////////
		//// Vaccum Pressures /////////
	   ///////////////////////////////
	   
M_UpdatePressureStates();

		 ///////////////////////////////
		////    Temperatures  /////////
	   ///////////////////////////////

// Master temperatrue to trigger sequences 

{IF defined (V1_HW)}

		 ///////////////////////////////////////
		//// Dew Point and ambiant temp ////
	   ///////////////////////////////////////

	stat.lrDewPointTempC := 	met_rh.rh_cry_wi.stat.lrDewPointTempC;
	stat.lrAmbiantTempC := 		met_temp.t_cry_wia.stat.lrTempC;
	stat.lrWindowMountTempC:= 	met_temp.t_cry_wim.stat.lrTempC;
	
	stat.lrDewPointTempK := 	met_rh.rh_cry_wi.stat.lrDewPointTempC + 273.15;
	stat.lrAmbiantTempK := 		met_temp.t_cry_wia.stat.lrTempK;
	stat.lrWindowMountTempK:= 	met_temp.t_cry_wim.stat.lrTempK;
	
	
	
		 ///////////////////////////////////////
		//// 		Cryo Temperatures 		////
	   ///////////////////////////////////////


	 stat.lrCryoTempK := met_temp.t_master.stat.lrTempK;
	 
	 stat.lrHighestTempK := met_temp.out_lrHighestTemp;
	 stat.lrLowestTempK	 := met_temp.out_lrLowestTemp;
	 stat.lrAverageOfAllTemps := met_temp.out_lrAverageOfAllTemps;
	 
	 stat.bHighestTempValid := met_temp.out_bHighestTempValid;
	 stat.bLowestTempValid := met_temp.out_bLowestTempValid; 
	 
	 stat.sHighestTempName := met_temp.out_sHighestTempName;
	 stat.sLowestTempName := met_temp.out_sLowestTempName;
(*
t_cry_Vote_1, t_cry_Vote_2, t_cry_Vote_3 temp votes are dedicated to estimate 
the temp of all three radiation shield segments.
t_cry_Vote_8 of cryo is dedicated to estimate the temperature of all shield segments
// TODO: Change the names in future
//	 
*) 
	 stat.lrRadShieldStiffRingTempK 	:=	met_temp.t_cry_vot_1.stat.lrTempK;	
	 stat.lrRadShieldIntermediateTempK 	:=	met_temp.t_cry_vot_2.stat.lrTempK;
	 stat.lrRadShieldBottomTempK		:=	met_temp.t_cry_vot_3.stat.lrTempK;
			
	 stat.lrRadiationShieldsTempK		:=	met_temp.t_cry_vot_8.stat.lrTempK;	
	 
 
{END_IF}
 
{IF defined (V2_SIM)}

		 ///////////////////////////////////////
		//// Dew Point and ambiant temp ////
	   ///////////////////////////////////////

	stat.lrDewPointTempC := 	sim_lrDewPointTempC;
	stat.lrAmbiantTempC := 		sim_lrAmbiantTempC;
	stat.lrWindowMountTempC:= 	sim_lrWindowMountTempC;
	
		 ///////////////////////////////////////
		//// 		Cryo Temperatures 		////
	   ///////////////////////////////////////


	 stat.lrCryoTempK := sim_lrCryostatTemp;
	 
	 stat.lrHighestTempK := sim_lrHighestTemp;
	 stat.lrLowestTempK	 := sim_lrLowestTemp;
	 stat.lrAverageOfAllTemps := 66.6;
	 
	 stat.bHighestTempValid := TRUE;
	 stat.bLowestTempValid := TRUE; 
	 
	 stat.sHighestTempName := 'Sim Highest Temp';
	 stat.sLowestTempName := 'Sim Lowest Temp';
	 
	 stat.lrRadiationShieldsTempK	:= sim_lrRadiationShielsTemp;

{END_IF}

bColdCond := stat.lrHighestTempK < cfg.lrTemp_Cold;
bWarmCond := stat.lrLowestTempK  > cfg.lrTemp_Warm;

trgCold(CLK := bColdCond);
trgWarm(CLK := bWarmCond);

(* Set flags based on conditions or trigger events *)
stat.bCold := bColdCond OR trgCold.Q;
stat.bWarm := bWarmCond OR trgWarm.Q;

(* Determine partial vacuum state when neither vacuum nor pressurized is active *)
stat.bPartiallyCold := (NOT stat.bCold) AND (NOT stat.bWarm);

		 ///////////////////////////////
		////    Interlocks  //////////
	   ///////////////////////////////
 

interlocks.bInterlock_Evacuation:=	   	 NOT ctrl.bSafe_Evac;		
interlocks.bInterlock_CoolDown:=		 NOT ctrl.bSafe_Cool_Down;	
interlocks.bInterlock_WarmUp:=			 NOT ctrl.bSafe_Warm_Up;	
interlocks.bInterlock_Regeneration:=	 NOT ctrl.bSafe_Regeneration;	
interlocks.bInterlock_AntiFogging:=		 NOT ctrl.bSafe_Anti_Fogging;

IF	stat.bEvacuationActive OR stat.bPumpsAreRunning THEN
	interlocks.bInterlock_Venting:= TRUE;
ELSE	   	 
	interlocks.bInterlock_Venting:= NOT ctrl.bSafe_Venting;
END_IF
///

met_venting.M_IsVentingFinishedSuccessfully(M_IsVentingFinishedSuccessfully => stat.bVentingFinishedSuccessfully);

		 ///////////////////////////////
		////    System Operational  //////////
	   ///////////////////////////////
	   
stat.bOP := met_cool_down.M_Get_ReadyForOperations();

		 ///////////////////////////////
		////    Interlocks  //////////
	   ///////////////////////////////
	   
	   	///////////////////////////////
		////    Stop PTCs  //////////
	   ///////////////////////////////
	   
stat.bStop_PTCs := met_warm_up.out_bStop_PTCs; 


	   	///////////////////////////////
		////    Local Time  //////////
	   ///////////////////////////////
END_METHOD

END_FUNCTION_BLOCK

// POUs/Devices/RH_Sensor/FB_METIS_RH
FUNCTION_BLOCK FB_METIS_RH
VAR_INPUT
END_VAR
VAR_OUTPUT
END_VAR
VAR_IN_OUT
	{attribute 'OPC.UA.DA' := '0'}
    met_temp : FB_METIS_TEMPERATURES;
END_VAR
VAR
    rh_cry_wi : FB_METIS_RH_SENSOR; // Relative Humidity sensor for the window
END_VAR


rh_cry_wi(in_sName := 'RH_CRY_WI', temperature := met_temp.t_cry_wia);

END_FUNCTION_BLOCK

// POUs/Devices/RH_Sensor/FB_METIS_RH_SENSOR
FUNCTION_BLOCK FB_METIS_RH_SENSOR EXTENDS FB_CRYO_SENSOR_BASE
VAR_INPUT
END_VAR
VAR_OUTPUT
END_VAR
VAR_IN_OUT
    temperature : FB_METIS_TEMPERATURE;
END_VAR
VAR
    // stat object
    stat : T_METIS_RH_SENSOR_STAT;    

    // command the digital output that powers the sensor
    power : FB_METIS_DO;
    
    // also run a dew point calculation
    dewPointCalc : FB_METIS_RH_DEWPOINT_CALC;
END_VAR

// set the reference
RefStat REF= stat;

// run the logic to operate the digital output
power(in_bInitialOutput := TRUE);

// run the sensor logic
SUPER^(in_sName := in_sName);

// run the dew point calculation
dewPointCalc(
    lrRhPercent         := stat.lrRhPercent,
    bRhValid            := stat.bValid,
    temperature         := temperature,
    lrDewPointTempC     => stat.lrDewPointTempC,
    bDewPointTempValid  => stat.bDewPointTempValid);

// Get input channel status and the raw reading
METHOD M_ReadSensor
VAR_INPUT
END_VAR
SUPER^.M_ReadSensor();

stat.lrRhFraction := INT_TO_LREAL(stat.nRawValue) / 32767;
stat.lrRhPercent  := stat.lrRhFraction * 100;
END_METHOD

METHOD M_SetStatus
VAR_INPUT
END_VAR
IF RefStat.bInputActive THEN
    RefStat.bValid 	        := TRUE; 
    RefStat.bError 	        := FALSE;
ELSE	
	RefStat.bValid	        := FALSE;
	RefStat.bError	        := TRUE;
END_IF
END_METHOD

END_FUNCTION_BLOCK

// POUs/Devices/DigitalOutput/FB_METIS_DO
FUNCTION_BLOCK FB_METIS_DO
VAR_INPUT
    in_bInitialOutput : BOOL;
END_VAR
VAR_OUTPUT
END_VAR
VAR
    {attribute 'OPC.UA.DA' := '1'}
    stat : T_METIS_DO_STAT;
    {attribute 'OPC.UA.DA' := '1'}
    ctrl : T_METIS_DO_CTRL;

    {attribute 'OPC.UA.DA' := '0'}
    bConfigured : BOOL;

    {attribute 'OPC.UA.DA' := '0'}
    i_nCouplerState     AT %I*: INT;
	{attribute 'OPC.UA.DA' := '0'}
	i_bOverTemperature  AT %I*: BOOL;
	{attribute 'OPC.UA.DA' := '0'}
    i_bOpenLoad         AT %I*: BOOL;
	{attribute 'OPC.UA.DA' := '0'}
    i_bOverCurrent      AT %I*: BOOL;
	{attribute 'OPC.UA.DA' := '0'}
    i_bShortCircuit     AT %I*: BOOL;
	{attribute 'OPC.UA.DA' := '0'}
	q_bOutput   AT %Q*: BOOL;
END_VAR

IF NOT bConfigured THEN
    M_Configure();
END_IF

// update the stat object
stat.bActive := ctrl.bEnable;
stat.bOpenLoad := i_bOpenLoad;
stat.bOverCurrent := i_bOverCurrent;
stat.bShortCircuit := i_bShortCircuit;
stat.bError := stat.bActive OR stat.bOpenLoad OR stat.bOverCurrent OR stat.bShortCircuit;

// update the output
q_bOutput := stat.bActive;

// update the status
M_UpdateStatus();

METHOD M_Configure : BOOL
VAR_INPUT
END_VAR
ctrl.bEnable := in_bInitialOutput;

bConfigured := TRUE;
END_METHOD

METHOD M_UpdateStatus
VAR_INPUT
END_VAR
IF i_nCouplerState <> 8 THEN
    stat.sStatus := 'Error: I/O not connected';
ELSIF stat.bOpenLoad THEN
    stat.sStatus := 'Error: open load';
ELSIF stat.bOverCurrent THEN
    stat.sStatus := 'Error: overcurrent';
ELSIF stat.bOverTemperature THEN
    stat.sStatus := 'Error: overtemperature';
ELSIF stat.bShortCircuit THEN
    stat.sStatus := 'Error: short circuit';
ELSIF stat.bError THEN
    stat.sStatus := 'ERROR';
ELSIF stat.bActive THEN
    stat.sStatus := 'ON';
ELSE
    stat.sStatus := 'OFF';
END_IF
END_METHOD

END_FUNCTION_BLOCK

// POUs/Devices/RH_Sensor/FB_METIS_RH_DEWPOINT_CALC
FUNCTION_BLOCK FB_METIS_RH_DEWPOINT_CALC
VAR_INPUT
    lrRhPercent : LREAL; // Relative humidity in percent, [0..100]
    bRhValid : BOOL; // TRUE if the lrHumidityPct value is valid
END_VAR
VAR_IN_OUT
    temperature : FB_METIS_TEMPERATURE;
END_VAR
VAR_OUTPUT
    lrDewPointTempC : LREAL;
    bDewPointTempValid : BOOL;
END_VAR
VAR
    
    out_lrDewPointTempK AT %Q* : LREAL;
    out_bDewPointTempValid  AT %Q* : BOOL;
END_VAR

bDewPointTempValid := bRhValid AND temperature.stat.bValid;

IF bDewPointTempValid THEN
    lrDewPointTempC := temperature.stat.lrTempC - ((100 - lrRhPercent)/5.0);
ELSE
    ; // don't update the last calculated dewpoint, i.e. keep the value frozen
END_IF

// update the outputs
out_lrDewPointTempK := lrDewPointTempC + 273.15;
out_bDewPointTempValid := bDewPointTempValid;

END_FUNCTION_BLOCK

// POUs/Devices/Temp_Voter/FB_METIS_VOTERS
FUNCTION_BLOCK FB_METIS_VOTERS
VAR_INPUT
END_VAR
VAR_OUTPUT
END_VAR
VAR_IN_OUT
	{attribute 'OPC.UA.DA' := '0'}
    met_temp : FB_METIS_TEMPERATURES;
END_VAR
VAR
	ctrl		: T_METIS_TEMP_VOTERS_CTRL;
    // CRY
	{attribute 'TcHmiSymbol.Show'}
    vote_cry_1  : FB_METIS_VOTER;
    vote_cry_2  : FB_METIS_VOTER;
    vote_cry_3  : FB_METIS_VOTER;
    vote_cry_4  : FB_METIS_VOTER;
    vote_cry_5  : FB_METIS_VOTER;
    vote_cry_6  : FB_METIS_VOTER;
    vote_cry_7  : FB_METIS_VOTER;
    vote_cry_8  : FB_METIS_VOTER;
    vote_cry_9  : FB_METIS_VOTER;
    vote_cry_10 : FB_METIS_VOTER;
    
    // SCA
    vote_sca_1  : FB_METIS_VOTER;
    vote_sca_2  : FB_METIS_VOTER;
    vote_sca_3  : FB_METIS_VOTER;
    vote_sca_4  : FB_METIS_VOTER;
    vote_sca_5  : FB_METIS_VOTER;
    vote_sca_6  : FB_METIS_VOTER;
    vote_sca_7  : FB_METIS_VOTER;
    vote_sca_8  : FB_METIS_VOTER;
    vote_sca_9  : FB_METIS_VOTER;
    vote_sca_10 : FB_METIS_VOTER;
    
    // IMG
    vote_img_1  : FB_METIS_VOTER;
    vote_img_2  : FB_METIS_VOTER;
    vote_img_3  : FB_METIS_VOTER;
    vote_img_4  : FB_METIS_VOTER;
    vote_img_5  : FB_METIS_VOTER;
    vote_img_6  : FB_METIS_VOTER;
    vote_img_7  : FB_METIS_VOTER;
    vote_img_8  : FB_METIS_VOTER;
    vote_img_9  : FB_METIS_VOTER;
    vote_img_10 : FB_METIS_VOTER;
	
	// System temperatures
	vote_master_temp	: FB_METIS_VOTER;
	vote_master_1		: FB_METIS_VOTER;
	vote_master_2		: FB_METIS_VOTER;
	
(************************
*** HMI *****************
************************)
// {attribute 'TcHmiSymbol.Show'}
// hmi_temp_vote_cry_1:	FB_METIS_HMI_CRYO_TEMPERATURE_VOTE;
// 
// //      TestIndexes : ARRAY[0..4] OF E_ALL_METIS_TEMPERATURES; 
// //  	TestMethod : E_METIS_TEMP_VOTE_METHOD; 


END_VAR

// CRY
vote_cry_1(in_sName  := 'VOTE_CRY_1', met_temp := met_temp);//, in_bSimulation := ctrl.tor_vote_cry_1.out_bEnable);//, bEnabled:= bEnableVoteCry1);
// vote_cry_2(in_sName  := 'VOTE_CRY_2', met_temp := met_temp);//, aTempIndexes := aVoteCry1TempIndexes, nVoteMethod := eVoteCry1Method, bEnabled := bEnableVoteCry1);
// vote_cry_3(in_sName  := 'VOTE_CRY_3', met_temp := met_temp);//, aTempIndexes := aVoteCry1TempIndexes, nVoteMethod := eVoteCry1Method, bEnabled := bEnableVoteCry1);
// vote_cry_4(in_sName  := 'VOTE_CRY_4', met_temp := met_temp);//, aTempIndexes := aVoteCry1TempIndexes, nVoteMethod := eVoteCry1Method, bEnabled := bEnableVoteCry1);
// vote_cry_5(in_sName  := 'VOTE_CRY_5', met_temp := met_temp);//, aTempIndexes := aVoteCry1TempIndexes, nVoteMethod := eVoteCry1Method, bEnabled := bEnableVoteCry1);
// vote_cry_6(in_sName  := 'VOTE_CRY_6', met_temp := met_temp);//, aTempIndexes := aVoteCry1TempIndexes, nVoteMethod := eVoteCry1Method, bEnabled := bEnableVoteCry1);
// vote_cry_7(in_sName  := 'VOTE_CRY_7', met_temp := met_temp);//, aTempIndexes := aVoteCry1TempIndexes, nVoteMethod := eVoteCry1Method, bEnabled := bEnableVoteCry1);
// vote_cry_8(in_sName  := 'VOTE_CRY_8', met_temp := met_temp);//, aTempIndexes := aVoteCry1TempIndexes, nVoteMethod := eVoteCry1Method, bEnabled := bEnableVoteCry1);
// vote_cry_9(in_sName  := 'VOTE_CRY_9', met_temp := met_temp);//, aTempIndexes := aVoteCry1TempIndexes, nVoteMethod := eVoteCry1Method, bEnabled := bEnableVoteCry1);
// vote_cry_10(in_sName:= 'VOTE_CRY_10', met_temp := met_temp);//, aTempIndexes := aVoteCry1TempIndexes, nVoteMethod := eVoteCry1Method, bEnabled := bEnableVoteCry1);
//                                                                                                                                
// // SCA                                                                                                                          
// vote_sca_1(in_sName  := 'VOTE_SCA_1', met_temp := met_temp);//, aTempIndexes := aVoteCry1TempIndexes, nVoteMethod := eVoteCry1Method, bEnabled := bEnableVoteCry1);
// vote_sca_2(in_sName  := 'VOTE_SCA_2', met_temp := met_temp);//, aTempIndexes := aVoteCry1TempIndexes, nVoteMethod := eVoteCry1Method, bEnabled := bEnableVoteCry1);
// vote_sca_3(in_sName  := 'VOTE_SCA_3', met_temp := met_temp);//, aTempIndexes := aVoteCry1TempIndexes, nVoteMethod := eVoteCry1Method, bEnabled := bEnableVoteCry1);
// vote_sca_4(in_sName  := 'VOTE_SCA_4', met_temp := met_temp);//, aTempIndexes := aVoteCry1TempIndexes, nVoteMethod := eVoteCry1Method, bEnabled := bEnableVoteCry1);
// vote_sca_5(in_sName  := 'VOTE_SCA_5', met_temp := met_temp);//, aTempIndexes := aVoteCry1TempIndexes, nVoteMethod := eVoteCry1Method, bEnabled := bEnableVoteCry1);
// vote_sca_6(in_sName  := 'VOTE_SCA_6', met_temp := met_temp);//, aTempIndexes := aVoteCry1TempIndexes, nVoteMethod := eVoteCry1Method, bEnabled := bEnableVoteCry1);
// vote_sca_7(in_sName  := 'VOTE_SCA_7', met_temp := met_temp);//, aTempIndexes := aVoteCry1TempIndexes, nVoteMethod := eVoteCry1Method, bEnabled := bEnableVoteCry1);
// vote_sca_8(in_sName  := 'VOTE_SCA_8', met_temp := met_temp);//, aTempIndexes := aVoteCry1TempIndexes, nVoteMethod := eVoteCry1Method, bEnabled := bEnableVoteCry1);
// vote_sca_9(in_sName  := 'VOTE_SCA_9', met_temp := met_temp);//, aTempIndexes := aVoteCry1TempIndexes, nVoteMethod := eVoteCry1Method, bEnabled := bEnableVoteCry1);
// vote_sca_10(in_sName:= 'VOTE_SCA_10', met_temp := met_temp);//, aTempIndexes := aVoteCry1TempIndexes, nVoteMethod := eVoteCry1Method, bEnabled := bEnableVoteCry1);
//                                                                                                                                
// // IMG                                                                                                                          
// vote_img_1(in_sName  := 'VOTE_IMG_1', met_temp := met_temp);//, aTempIndexes := aVoteCry1TempIndexes, nVoteMethod := eVoteCry1Method, bEnabled := bEnableVoteCry1);
// vote_img_2(in_sName  := 'VOTE_IMG_2', met_temp := met_temp);//, aTempIndexes := aVoteCry1TempIndexes, nVoteMethod := eVoteCry1Method, bEnabled := bEnableVoteCry1);
// vote_img_3(in_sName  := 'VOTE_IMG_3', met_temp := met_temp);//, aTempIndexes := aVoteCry1TempIndexes, nVoteMethod := eVoteCry1Method, bEnabled := bEnableVoteCry1);
// vote_img_4(in_sName  := 'VOTE_IMG_4', met_temp := met_temp);//, aTempIndexes := aVoteCry1TempIndexes, nVoteMethod := eVoteCry1Method, bEnabled := bEnableVoteCry1);
// vote_img_5(in_sName  := 'VOTE_IMG_5', met_temp := met_temp);//, aTempIndexes := aVoteCry1TempIndexes, nVoteMethod := eVoteCry1Method, bEnabled := bEnableVoteCry1);
// vote_img_6(in_sName  := 'VOTE_IMG_6', met_temp := met_temp);//, aTempIndexes := aVoteCry1TempIndexes, nVoteMethod := eVoteCry1Method, bEnabled := bEnableVoteCry1);
// vote_img_7(in_sName  := 'VOTE_IMG_7', met_temp := met_temp);//, aTempIndexes := aVoteCry1TempIndexes, nVoteMethod := eVoteCry1Method, bEnabled := bEnableVoteCry1);
// vote_img_8(in_sName  := 'VOTE_IMG_8', met_temp := met_temp);//, aTempIndexes := aVoteCry1TempIndexes, nVoteMethod := eVoteCry1Method, bEnabled := bEnableVoteCry1);
// vote_img_9(in_sName  := 'VOTE_IMG_9', met_temp := met_temp);//, aTempIndexes := aVoteCry1TempIndexes, nVoteMethod := eVoteCry1Method, bEnabled := bEnableVoteCry1);
// vote_img_10(in_sName:= 'VOTE_IMG_10', met_temp := met_temp);//, aTempIndexes := aVoteCry1TempIndexes, nVoteMethod := eVoteCry1Method, bEnabled := bEnableVoteCry1);
// 
// // System temperatures
// vote_master_temp(in_sName := 'MASTER_TEMP',   met_temp := met_temp);//, aTempIndexes := aVoteCry1TempIndexes, nVoteMethod := eVoteCry1Method, bEnabled := bEnableVoteCry1);
// vote_master_1(in_sName    := 'VOTE_MASTER_1', met_temp := met_temp);//, aTempIndexes := aVoteCry1TempIndexes, nVoteMethod := eVoteCry1Method, bEnabled := bEnableVoteCry1);
// vote_master_2(in_sName    := 'VOTE_MASTER_2', met_temp := met_temp);//, aTempIndexes := aVoteCry1TempIndexes, nVoteMethod := eVoteCry1Method, bEnabled := bEnableVoteCry1);

M_ReadSensors();

M_ProcessHmi();

METHOD M_ProcessHmi : BOOL
VAR_INPUT
END_VAR
// hmi_temp_vote_cry_1(
// 	inout_sTemperatureStatRef 	:= vote_cry_1.stat,
// 	inout_sCmdOver 				:= ctrl.tor_vote_cry_1,
// 	inout_fbAlarmHandlerRef 	:= vote_cry_1.fbAlarmHandler,
// //	TestIndexes := TestIndexes, TestMethod := TestMethod
// );
END_METHOD

METHOD M_ReadSensors : BOOL
VAR_INPUT
END_VAR
//
// Read temperature votes.
//
// Execute Temperature Override (tor) of simulation flags.
ctrl.tor_vote_cry_1(in_bEnable:=ctrl.bSim_Temp_vote_cry_1);
END_METHOD

END_FUNCTION_BLOCK

// POUs/Devices/Temp_Voter/FB_METIS_VOTER
FUNCTION_BLOCK FB_METIS_VOTER
VAR_INPUT
	{attribute 'OPC.UA.DA' := '0'}
	in_sName:	STRING;
// 	{attribute 'OPC.UA.DA' := '0'}
// 	in_bSimulation	: BOOL;
	{attribute 'OPC.UA.DA' := '0'}
	in_nRampPeriodSec:		UDINT := 60;	// Ramp measurement period [sec]. Default 60 sec.
END_VAR
VAR_IN_OUT
	{attribute 'OPC.UA.DA' := '0'}
	met_temp: FB_METIS_TEMPERATURES;
END_VAR
VAR
	cfg:				T_METIS_TEMP_VOTE_CFG;
// 	{attribute 'OPC.UA.DA' := '0'}
// 	bSimulation	: BOOL := FALSE;	// Simulated temp value

	{attribute 'OPC.UA.DA' := '0'}
	aTempPointers:	    ARRAY[0..4] OF POINTER TO FB_METIS_TEMPERATURE;
	{attribute 'OPC.UA.DA' := '0'}
	aTempIndexes:		ARRAY[0..4] OF INT := [0, 0, 0, 0, 0];
	
	(*Voting Method*)
	nVoteMethod:	E_METIS_TEMP_VOTE_METHOD := E_METIS_TEMP_VOTE_METHOD.AVERAGE;

	{attribute 'TcHmiSymbol.Show'}
	{attribute 'OPC.UA.DA' := '1'}
	stat	: T_METIS_CRYO_TEMP_VOTE_STATUS;
    
    (* OLD PLC_HMI  *)
	{attribute 'TcHmiSymbol.Show'}
    bPLC_HMI:       BOOL := FALSE;
    
    (* User description *)
    //sDescription:   STRING;
    
	(*Engineering MODE*)
	{attribute 'TcHmiSymbol.Show'}
	bEngMode:		BOOL := FALSE;
	{attribute 'TcHmiSymbol.Show'}
	bAutoMode:		BOOL := TRUE;
	{attribute 'TcHmiSymbol.Show'}
	bManualMode:	BOOL := FALSE;	

	(*Configuration*)
	bConfigured:	BOOL := FALSE;
	
	(*Read/Write configuration*)
	{attribute 'OPC.UA.DA' := '0'}
	{attribute 'TcHmiSymbol.Show'}
	fbTempVoteConfig:		FB_READ_WRITE_TEMP_VOTE_CONFIG;
	{attribute 'TcHmiSymbol.Show'}
	bReadConfig:			BOOL;
	{attribute 'TcHmiSymbol.Show'}	
	bWriteConfig:			BOOL;
	(*Ramp *)
	{attribute 'OPC.UA.DA' := '0'}
	bRampTimerStarted:	BOOL := FALSE;
	{attribute 'OPC.UA.DA' := '0'}
	rampTimer:	TON;		// Timer for calculating ramp
	
    // outputs that can be used for linking
	{attribute 'OPC.UA.DA' := '0'}
    q_lrTemp    AT %Q*: LREAL;
	{attribute 'OPC.UA.DA' := '0'}
	q_bToggle   AT %Q*: BOOL;
	{attribute 'OPC.UA.DA' := '0'}
	q_bValid   AT %Q*: BOOL := FALSE;
	
	{attribute 'TcHmiSymbol.Show'}
	{attribute 'TcHmiSymbol.ReadOnly'}
	sEventClassName : T_MaxString;


	{attribute 'TcHmiSymbol.Show'}
	bConfirmAllAlarms : BOOL;
	
		// Alarm handling
	// List of alarms to be handled by Temperature
	arrEventEntry : ARRAY [0..5] OF TcEventEntry;
	// Alarm handler FB

	fbAlarmHandler : FB_AlarmHandler;
	{attribute 'TcHmiSymbol.Show'}
	{attribute 'TcHmiSymbol.ReadOnly'}
	sInstanceName : T_MaxString := fbAlarmHandler.sInstanceName;
	// Logs logs
	logs:	FB_CRYO_FUNCTION_LOG;
END_VAR

// to avoid any problem of invalid pointers, set them right away
M_UpdateTempPointers(met_temp := met_temp);

(*Read/Write configuration*)
fbTempVoteConfig(in_sTVoteName:= in_sName, Temp_Vote_Config:= cfg);

IF NOT bConfigured THEN
    M_Configure(met_temp := met_temp);
    RETURN;
END_IF

// set AUTO / MAN / ENG
M_SetPermissionMode();

// read/write the config (if needed)
M_Read_Write_Config(met_temp := met_temp);

M_GetRamp();

M_SetStatus();


// Handle alarms
M_UpdateAlarms();

PROPERTY bTempNotValid : BOOL
GET
bTempNotValid := NOT stat.bValid;
END_GET
END_PROPERTY

PROPERTY bTempValid : BOOL
GET
bTempValid := stat.bValid;
END_GET
END_PROPERTY

PROPERTY lrRamp : LREAL
GET
lrRamp := stat.lrRamp;
END_GET
END_PROPERTY

PROPERTY lrTempK : LREAL
GET
lrTempK := stat.lrTempK;
END_GET
END_PROPERTY

METHOD M_ConfigReadingFinished
VAR_INPUT
    bError : BOOL;
END_VAR
VAR_IN_OUT
    met_temp : FB_METIS_TEMPERATURES;
END_VAR
VAR
    i : INT;
END_VAR
IF bError THEN
   // ERROR! Just put the indexes to 0
   FOR i := 0 TO 4 DO
       aTempIndexes[i] := 0;
   END_FOR
   stat.bEnabled := FALSE;
   stat.sDescription := in_sName;
ELSE
    // success!
//     aTempIndexes[0] := met_temp.M_GetTempSensorIndex(cfg.sTemp1_Name);
//     aTempIndexes[1] := met_temp.M_GetTempSensorIndex(cfg.sTemp2_Name);
//     aTempIndexes[2] := met_temp.M_GetTempSensorIndex(cfg.sTemp3_Name);
//     aTempIndexes[3] := met_temp.M_GetTempSensorIndex(cfg.sTemp4_Name);
//     aTempIndexes[4] := met_temp.M_GetTempSensorIndex(cfg.sTemp5_Name);
// 	aTempIndexes[0] 	:= TO_INT(cfg.eTemperature1);
// 	aTempIndexes[1] 	:= TO_INT(cfg.eTemperature2);
// 	aTempIndexes[2] 	:= TO_INT(cfg.eTemperature3);
// 	aTempIndexes[3] 	:= TO_INT(cfg.eTemperature4);
// 	aTempIndexes[4] 	:= TO_INT(cfg.eTemperature5);
    stat.nVoteMethod     := cfg.nVote_Method;
    stat.bEnabled        := cfg.bEnabled;
    stat.sDescription    := cfg.sDescription;
	stat.aTempIndexes[0] := cfg.eTemperature1;
	stat.aTempIndexes[1] := cfg.eTemperature2;
    stat.aTempIndexes[2] := cfg.eTemperature3;
	stat.aTempIndexes[3] := cfg.eTemperature4;
    stat.aTempIndexes[4] := cfg.eTemperature5; 
END_IF

M_UpdateTempPointers(met_temp := met_temp);

// clear the flag
fbTempVoteConfig.M_ClearReadingDoneFlag();
END_METHOD

METHOD M_Configure : BOOL
VAR_INPUT
END_VAR
VAR_INST
	{attribute 'OPC.UA.DA' := '0'}
    nConfigureState : INT;
END_VAR
VAR_IN_OUT
	{attribute 'OPC.UA.DA' := '0'}
    met_temp : FB_METIS_TEMPERATURES;
END_VAR
VAR
    i : INT;
END_VAR











CASE nConfigureState OF
    0:  
        // use the name of the voter as the default description
        stat.sDescription := in_sName;
        // start reading the config
        fbTempVoteConfig.M_ReadConfiguration();
        nConfigureState := 1;
    1:
        IF fbTempVoteConfig.bReadingDoneFlag THEN
            M_ConfigReadingFinished(
                bError   := fbTempVoteConfig.bReadError,
                met_temp := met_temp);
		
			//
	// Populate array of Alarms.
	//
	// See the definition of CryoPressVoteEventClass under Type System.
	//
	arrEventEntry[0] := Tc_Events.METISCryoTempEventClass.ReadingNotValid;
	arrEventEntry[1] := Tc_Events.METISCryoTempEventClass.Sensor1Error;
	arrEventEntry[2] := Tc_Events.METISCryoTempEventClass.Sensor2Error;
	arrEventEntry[3] := Tc_Events.METISCryoTempEventClass.Sensor3Error;
	arrEventEntry[4] := Tc_Events.METISCryoTempEventClass.Sensor4Error;
	arrEventEntry[5] := Tc_Events.METISCryoTempEventClass.Sensor5Error;
            
            bConfigured := TRUE;
        END_IF
END_CASE
END_METHOD

METHOD M_GetRamp
VAR_INPUT
END_VAR
VAR_INST
	{attribute 'OPC.UA.DA' := '0'}
	lrRampStartTempK:	LREAL;	// Temperature at start of ramp timer [K]
END_VAR
VAR
	nRampPeriodSec:		UDINT;	// Ramp measurement period [sec].
END_VAR

IF NOT (stat.bEnabled AND stat.bValid) THEN
    bRampTimerStarted := FALSE;
    stat.lrRamp := 0.0;
    RETURN;
END_IF

IF NOT bRampTimerStarted THEN
	bRampTimerStarted	:= TRUE;
	lrRampStartTempK	:= stat.lrTempK;
	rampTimer(IN:=FALSE);
END_IF

// Execute timer.
// Ramp measurement period should be > 0
nRampPeriodSec	:= in_nRampPeriodSec;
IF nRampPeriodSec = 0 THEN
	nRampPeriodSec	:= 60;
END_IF
rampTimer(IN:=TRUE,PT:=UDINT_TO_TIME(nRampPeriodSec)*1000);

// Calculate ramp at time expiry
IF rampTimer.Q THEN
	// Calculate the temperature ramp per minute
//	IF stat.bValid THEN
		stat.lrRamp	:= (stat.lrTempK - lrRampStartTempK) * 60.0 / nRampPeriodSec;
//	ELSE
//		stat.lrRamp	:= 0.0;
//	END_IF

	// Current temperature is the starting value of the ramp
	lrRampStartTempK	:= stat.lrTempK;

	// Restart the timer
	rampTimer(IN:=FALSE);
END_IF
END_METHOD

METHOD M_Read_Write_Config
VAR_INPUT
END_VAR
VAR_IN_OUT
    met_temp : FB_METIS_TEMPERATURES;
END_VAR
IF bEngMode THEN
    IF bWriteConfig THEN
        
        // update the cfg object
        cfg.bEnabled     := stat.bEnabled;
        cfg.sDescription := stat.sDescription;
        cfg.sTemp1_Name  := aTempPointers[0]^.in_sName;
        cfg.sTemp2_Name  := aTempPointers[1]^.in_sName; 
        cfg.sTemp3_Name  := aTempPointers[2]^.in_sName; 
        cfg.sTemp4_Name  := aTempPointers[3]^.in_sName; 
        cfg.sTemp5_Name  := aTempPointers[4]^.in_sName;
        cfg.nVote_Method := stat.nVoteMethod;
		cfg.eTemperature1:= stat.aTempIndexes[0];
		cfg.eTemperature2:= stat.aTempIndexes[1];
		cfg.eTemperature3:= stat.aTempIndexes[2];
		cfg.eTemperature4:= stat.aTempIndexes[3];
		cfg.eTemperature5:= stat.aTempIndexes[4];
        
        // write the cfg object
        fbTempVoteConfig.M_WriteConfiguration();
        bWriteConfig := FALSE;
                
    ELSIF bReadConfig THEN
	
        fbTempVoteConfig.M_ReadConfiguration();
        bReadConfig := FALSE;
        
    END_IF
		
END_IF

IF fbTempVoteConfig.bReadingDoneFlag THEN
	M_ConfigReadingFinished(
        bError := fbTempVoteConfig.bReadError,
        met_temp := met_temp);
END_IF
END_METHOD

METHOD M_SetPermissionMode : BOOL
VAR_INPUT
END_VAR
IF bAutoMode THEN
    stat.sStatus    := 'AUTO';
    bManualMode     := FALSE;
    bEngMode        := FALSE;
ELSIF bEngMode	THEN
    stat.sStatus    := 'ENG';
    bManualMode     := FALSE;
    bAutoMode       := FALSE;
ELSIF bManualMode THEN
    stat.sStatus    := 'MANUAL';
    bAutoMode       := FALSE;
    bEngMode        := FALSE;
END_IF
END_METHOD

// Calculate pressure based on the status of the two sensors
METHOD M_SetStatus
VAR_INPUT
END_VAR
VAR
	lrTmp:		LREAL;	// Temporary var
	nSample:	INT;
	i:			INT;
END_VAR
VAR_INST
	{attribute 'OPC.UA.DA' := '0'}
    toggleTimer : TON;
END_VAR
aTempIndexes[0] 	:= TO_INT(stat.aTempIndexes[0]);
aTempIndexes[1] 	:= TO_INT(stat.aTempIndexes[1]);
aTempIndexes[2] 	:= TO_INT(stat.aTempIndexes[2]);
aTempIndexes[3] 	:= TO_INT(stat.aTempIndexes[3]);
aTempIndexes[4] 	:= TO_INT(stat.aTempIndexes[4]);


stat.lrSens1TempK := aTempPointers[0]^.stat.lrTempK;
stat.lrSens2TempK := aTempPointers[1]^.stat.lrTempK;
stat.lrSens3TempK := aTempPointers[2]^.stat.lrTempK;
stat.lrSens4TempK := aTempPointers[3]^.stat.lrTempK;
stat.lrSens5TempK := aTempPointers[4]^.stat.lrTempK;

stat.bValidSensor1  := aTempPointers[0]^.stat.bValid;
stat.bValidSensor2  := aTempPointers[1]^.stat.bValid;
stat.bValidSensor3  := aTempPointers[2]^.stat.bValid;
stat.bValidSensor4  := aTempPointers[3]^.stat.bValid;
stat.bValidSensor5  := aTempPointers[4]^.stat.bValid;

// copy some writeable values to the read-only stat struct
//stat.bEnabled := bEnabled;
//stat.sDescription := sDescription;

sInstanceName := fbAlarmHandler.sInstanceName;
sEventClassName := fbAlarmHandler.sEventClassName;
IF bConfirmAllAlarms THEN
	bConfirmAllAlarms := FALSE;
	fbAlarmHandler.M_ConfirmAllAlarms();
END_IF


// If disabled, don't do anything
IF NOT stat.bEnabled THEN
    stat.bValid := FALSE;
    RETURN;
END_IF

//
// If simulated, set the simulated value and return.
//
IF stat.bSimulated THEN
// 	stat.bSimulated	:= TRUE;
	stat.bValid		:= TRUE;
	stat.lrTempK	:= stat.lrSimTempK;
	RETURN;
ELSE
	stat.bSimulated	:= FALSE;
END_IF


//
// Get the pressure depending on the voting method.
//
CASE nVoteMethod OF
	E_METIS_TEMP_VOTE_METHOD.AVERAGE:
		M_SetStatus_Average();
	E_METIS_TEMP_VOTE_METHOD.LOWEST_TEMPERATURE:
		M_SetStatus_Lowest_Temperature();
	E_METIS_TEMP_VOTE_METHOD.HIGHEST_TEMPERATURE:
		M_SetStatus_Highest_Temperature();
	E_METIS_TEMP_VOTE_METHOD.FIRST_VALID_TEMPERATURE:
		M_SetStatus_FirstValid();
	E_METIS_TEMP_VOTE_METHOD.MEDIAN:
		M_SetStatus_Median();
//	E_METIS_TEMP_VOTE_METHOD.TEMPERATURE_3oo5:
//		M_SetStatus_XooY();
ELSE
	;
END_CASE


//
// If the reading is valid, set the simulated value to it.
// This way, switching from normal to simulation will result in
// no jump in the value.
//
IF stat.bValid  THEN
	stat.lrSimTempK	:= stat.lrTempK;
END_IF

// update also the output data
q_lrTemp := stat.lrTempK;
q_bValid := stat.bValid;
toggleTimer(IN := NOT toggleTimer.Q, PT := T#500ms);
IF toggleTimer.Q AND stat.bValid THEN
    q_bToggle := NOT q_bToggle;
END_IF
END_METHOD

METHOD M_SetStatus_Average
VAR_INPUT
END_VAR
VAR
	lrTmp:		LREAL;	// Temporary var for sum of Temperatures
	nSample:	INT;	// Number of valid sensor readings
	i:			INT;
END_VAR
lrTmp	:= 0.0;
nSample	:= 0;

FOR i:=0 TO 4 DO
	IF aTempIndexes[i] > 0  THEN
		IF aTempPointers[i]^.stat.bValid	THEN
			lrTmp	:= lrTmp + aTempPointers[i]^.stat.lrTempK;
			nSample	:= nSample + 1;
		END_IF
	END_IF
END_FOR

IF nSample > 0	THEN
	stat.lrTempK	:= lrTmp / nSample;
	stat.bValid		:= TRUE;
ELSE
	stat.lrTempK	:= 9999;
	stat.bValid		:= FALSE;
END_IF
END_METHOD

METHOD M_SetStatus_FirstValid
VAR_INPUT
END_VAR
VAR
	lrTmp:		LREAL;	// Temporary var for sum of Temperatures
	nSample:	INT;	// Number of valid sensor readings
	i:			INT;
END_VAR
(*First Valid Temperature*)

nSample	:= 0;

FOR i:=0 TO 4 DO
	IF aTempIndexes[i] > 0  THEN
		IF  aTempPointers[i]^.stat.bValid	THEN
			lrTmp	:= aTempPointers[i]^.stat.lrTempK;
			nSample	:= nSample + 1;
			EXIT;
		END_IF
	END_IF
END_FOR

IF nSample > 0	THEN
	stat.lrTempK	:= lrTmp;
	stat.bValid		:= TRUE;
ELSE
	stat.lrTempK	:= 9999;
	stat.bValid		:= FALSE;
END_IF
END_METHOD

METHOD M_SetStatus_Highest_Temperature
VAR_INPUT
END_VAR
VAR
	lrTmp:		LREAL;	// Temporary var for sum of Temperatures
	nSample:	INT;	// Number of valid sensor readings
	i:			INT;
END_VAR
(*Highest Temperature*)

lrTmp	:= -10000.0; // setting initial temperature for comparision
nSample	:= 0;

FOR i:=0 TO 4 DO
	IF aTempIndexes[i] > 0  THEN
		IF  aTempPointers[i]^.stat.bValid	THEN
				IF  aTempPointers[i]^.stat.lrTempK > lrTmp THEN
					lrTmp	:= aTempPointers[i]^.stat.lrTempK;
				END_IF
			nSample	:= nSample + 1;
		END_IF
	END_IF
END_FOR

IF nSample > 0	THEN
	stat.lrTempK	:= lrTmp;
	stat.bValid		:= TRUE;
ELSE
	stat.lrTempK	:= 9999;
	stat.bValid		:= FALSE;
END_IF
END_METHOD

METHOD M_SetStatus_Lowest_Temperature
VAR_INPUT
END_VAR
VAR
	lrTmp:		LREAL;	// Temporary var for sum of Temperatures
	nSample:	INT;	// Number of valid sensor readings
	i:			INT;
END_VAR
(*Lowest Temperature*)

lrTmp	:= 10000.0; // setting initial temperature for comparision
nSample	:= 0;

FOR i:=0 TO 4 DO
	IF aTempIndexes[i] > 0  THEN
		IF  aTempPointers[i]^.stat.bValid	THEN
				IF  aTempPointers[i]^.stat.lrTempK < lrTmp THEN
					lrTmp	:= aTempPointers[i]^.stat.lrTempK;
				END_IF
			nSample	:= nSample + 1;
		END_IF
	END_IF
END_FOR

IF nSample > 0	THEN
	stat.lrTempK	:= lrTmp;
	stat.bValid		:= TRUE;
ELSE
	stat.lrTempK	:= 9999;
	stat.bValid		:= FALSE;
END_IF
END_METHOD

METHOD M_SetStatus_Median
VAR_INPUT
END_VAR
VAR
    lrTmpArray: ARRAY[0..4] OF LREAL; // Array to store valid temperatures
    nSample:    INT;                // Number of valid sensor readings
    i:          INT;
    j:          INT;
    lrTemp:     LREAL;             // Temporary variable for swapping
END_VAR
nSample := 0;

// Store valid temperatures in the array
FOR i := 0 TO 4 DO
    IF aTempIndexes[i] > 0 THEN
        IF aTempPointers[i]^.stat.bValid THEN
            lrTmpArray[nSample] := aTempPointers[i]^.stat.lrTempK;
            nSample := nSample + 1;
        END_IF
    END_IF
END_FOR

// Sort the array in ascending order (using Bubble Sort for simplicity)
IF nSample > 1 THEN
    FOR i := 0 TO nSample - 2 DO
        FOR j := i + 1 TO nSample - 1 DO
            IF lrTmpArray[i] > lrTmpArray[j] THEN
                lrTemp := lrTmpArray[i];
                lrTmpArray[i] := lrTmpArray[j];
                lrTmpArray[j] := lrTemp;
            END_IF
        END_FOR
    END_FOR
END_IF

// Calculate the median
IF nSample > 0 THEN
    IF nSample MOD 2 = 1 THEN // Odd number of elements
        stat.lrTempK := lrTmpArray[nSample / 2];
    ELSE // Even number of elements
        stat.lrTempK := (lrTmpArray[nSample / 2 - 1] + lrTmpArray[nSample / 2]) / 2.0;
    END_IF
    stat.bValid := TRUE;
ELSE
    stat.lrTempK := 9999;
    stat.bValid := FALSE;
END_IF
END_METHOD

// Calculate pressure based on the status of the two sensors
METHOD M_SetStatus_XooY
//VAR_INPUT
//	in_nNum:	INT;	// Number of readings to select for voting (X)
//	in_nTotal:	INT;	// Total number of readings to check (Y)
//END_VAR
//VAR
//	idx_i, idx_j:	INT;
//	nTmp:		INT;			// Temporary INT var
//	lrTmp:		LREAL	:= 0.0;	// Temporary var for sum of pressures
//	nValid:		INT		:= 0;	// Total number of valid readings
//	nSample:	INT		:= 0;	// Number of valid sensor readings
	
//	aDiff:		ARRAY [1..5,1..5] OF LREAL;	// Table of absolute differences
//	aDiffSum:	ARRAY [1..5] OF LREAL;		// Array of sums of absolute differences
//	// Array of indexes of sums of absolute differences
//	aDiffSumIdx:ARRAY [1..5] OF INT := [1,2,3,4,5];		
//	lrAbsDiff:	LREAL;						// Absolute difference between two readings
	
//	i:			INT;
//	j:			INT;
//END_VAR
VAR
	lrTmp:		LREAL;	// Temporary var for sum of Temperatures
	nSample:	INT;	// Number of valid sensor readings
	i:			INT;
END_VAR
(*Average Temperature*)

lrTmp	:= 0.0;
nSample	:= 0;

FOR i:=0 TO 4 DO
	IF aTempIndexes[i] > 0  THEN
		IF  aTempPointers[i]^.stat.bValid	THEN
			lrTmp	:= lrTmp + aTempPointers[i]^.stat.lrTempK;
			nSample	:= nSample + 1;
		END_IF
	END_IF
END_FOR

IF nSample > 0	THEN
	stat.lrTempK	:= lrTmp / nSample;
	stat.bValid		:= TRUE;
ELSE
	stat.lrTempK	:= 9999;
	stat.bValid		:= FALSE;
END_IF








////
////	Get the number of valid readings and calculate the average
////
//FOR i:=1 TO in_nTotal DO
//	IF pSensor[i] <> 0  THEN
//		IF  pSensor[i]^.stat.bValid	THEN
//			lrTmp	:= lrTmp + pSensor[i]^.stat.lrPressure;
//			nValid	:= nValid + 1;
//		END_IF
//	END_IF
//END_FOR


////
//// Vote X out of Y
////
//IF nValid >= in_nNum	THEN
//	//
//	// Calculate relative differences between two readings, 
//	// relative to the bigger ABS value.
//	// Table is symetric. Calculate only the half (triangle) on the right. 
//	// Make a copy to the other half.
//	//
//	FOR i:=1 TO in_nTotal DO
//		FOR j:=i+1 TO in_nTotal DO
//			IF pSensor[i] <> 0  AND  pSensor[j] <> 0	THEN
//				IF pSensor[i]^.stat.bValid  AND  pSensor[j]^.stat.bValid	THEN
//					lrAbsDiff	:= ABS(pSensor[i]^.stat.lrPressure - pSensor[j]^.stat.lrPressure);
//					aDiff[i,j]	:= lrAbsDiff;
//					aDiff[j,i]	:= lrAbsDiff;
//				ELSE
//					aDiff[i,j]	:= 9999.0;
//					aDiff[j,i]	:= 9999.0;
//				END_IF
//			ELSE
//				aDiff[i,j]	:= 9999.0;
//				aDiff[j,i]	:= 9999.0;
//			END_IF
//		END_FOR
//	END_FOR

//	//
//	// Get the sum of all differences for each reading.
//	//
//	FOR i:=1 TO in_nTotal DO
//		aDiffSum[i]	:= 0.0;
//		FOR j:=1 TO in_nTotal DO
//			aDiffSum[i]	:= aDiffSum[i] + aDiff[i,j];
//		END_FOR
//	END_FOR

//	//
//	// Sort the indexes for differences in accending order (low sum first).
//	//
//	FOR i:=1 TO in_nTotal DO
//		FOR j:=i+1 TO in_nTotal DO
//			idx_i	:= aDiffSumIdx[i];
//			idx_j	:= aDiffSumIdx[j];
//			IF aDiffSum[idx_j] < aDiffSum[idx_i]	THEN
//				// Swap indexes
//				nTmp			:= aDiffSumIdx[j];
//				aDiffSumIdx[j]	:= aDiffSumIdx[i];
//				aDiffSumIdx[i]	:= nTmp;
//			END_IF
//		END_FOR
//	END_FOR

	
//	//					
//	// Get the average of selected in_nNum readings.
//	// Assign the result to the pressure.
//	//
//	lrTmp	:= 0.0;
//	FOR i:=1 TO in_nNum DO
//		idx_i	:= aDiffSumIdx[i];
//		lrTmp	:= lrTmp + pSensor[idx_i]^.stat.lrPressure;
//	END_FOR
	
//	stat.lrPressure	:= lrTmp / in_nNum;
//	stat.bValid		:= TRUE;
//ELSE
//	stat.lrPressure	:= 9999;
//	stat.bValid		:= FALSE;
//END_IF
END_METHOD

METHOD M_UpdateAlarms
VAR_INPUT
END_VAR
VAR
	stEventEntry : TcEventEntry;
	sText : STRING;
END_VAR
//
// Set / clear alarms
//

// Global alarm if the voted temperature reading is not valid.
fbAlarmHandler.M_UpdateAlarm(
    in_bCondition    := NOT stat.bValid,
    in_nIndex        := 0,
    in_strEventEntry := Tc_Events.METISCryoTempEventClass.ReadingNotValid
);


// Individual sensor alarms.
// Important:
// Even if aTempIndexes[x] = 0, M_UpdateAlarm is still called with FALSE.
// This ensures that any previously active alarm is cleared automatically.

fbAlarmHandler.M_UpdateAlarm(
    in_bCondition    := (aTempIndexes[0] > 0) AND (NOT aTempPointers[0]^.stat.bValid),
    in_nIndex        := 1,
    in_strEventEntry := Tc_Events.METISCryoTempEventClass.Sensor1Error
);

fbAlarmHandler.M_UpdateAlarm(
    in_bCondition    := (aTempIndexes[1] > 0) AND (NOT aTempPointers[1]^.stat.bValid),
    in_nIndex        := 2,
    in_strEventEntry := Tc_Events.METISCryoTempEventClass.Sensor2Error
);

fbAlarmHandler.M_UpdateAlarm(
    in_bCondition    := (aTempIndexes[2] > 0) AND (NOT aTempPointers[2]^.stat.bValid),
    in_nIndex        := 3,
    in_strEventEntry := Tc_Events.METISCryoTempEventClass.Sensor3Error
);

fbAlarmHandler.M_UpdateAlarm(
    in_bCondition    := (aTempIndexes[3] > 0) AND (NOT aTempPointers[3]^.stat.bValid),
    in_nIndex        := 4,
    in_strEventEntry := Tc_Events.METISCryoTempEventClass.Sensor4Error
);

fbAlarmHandler.M_UpdateAlarm(
    in_bCondition    := (aTempIndexes[4] > 0) AND (NOT aTempPointers[4]^.stat.bValid),
    in_nIndex        := 5,
    in_strEventEntry := Tc_Events.METISCryoTempEventClass.Sensor5Error
);


//
// Handle alarms
//
fbAlarmHandler(stAlarms := stat.stAlarms);

fbAlarmHandler.M_ProcessAlarms(
    arrEventEntry := arrEventEntry,
    sEventString  := in_sName
);
END_METHOD

METHOD M_UpdateTempPointers
VAR_INPUT
END_VAR
VAR_IN_OUT
    met_temp : FB_METIS_TEMPERATURES;
END_VAR
VAR 
    i : INT;
END_VAR
// FOR i := 0 TO 4 DO
//     aTempPointers[i] := met_temp.M_SetTemperatureSensor(aTempIndexes[i]);
// END_FOR

FOR i := 0 TO 4 DO
	IF bPLC_HMI THEN
	    aTempPointers[i] := met_temp.M_SetTemperatureSensor(TO_INT(aTempIndexes[i]));
	ELSE	(*Temp selection from new HMI*)
    	aTempPointers[i] := met_temp.M_SetTemperatureSensor(TO_INT(stat.aTempIndexes[i]));
	END_IF


END_FOR
END_METHOD

END_FUNCTION_BLOCK

// POUs/XML_Cfg_Read_Write/FB_READ_WRITE_TEMP_VOTE_CONFIG
FUNCTION_BLOCK FB_READ_WRITE_TEMP_VOTE_CONFIG EXTENDS FB_READ_WRITE_CONFIG_BASE
VAR_INPUT
	in_sTVoteName:      T_MaxString;
END_VAR
VAR_IN_OUT
	Temp_Vote_Config:   T_METIS_TEMP_VOTE_CFG;
END_VAR

SUPER^(
    in_sEntryName  := in_sTVoteName,
    in_sSubFolder  := 'Temperature_Vote\',
    in_sXPath      := '/Temperature_Vote_Configuration/',
    in_pSymAddr    := ADR(Temp_Vote_Config),
    in_cbSymSize   := SIZEOF(Temp_Vote_Config));

END_FUNCTION_BLOCK

// HMIWrapperFBs/FB_METIS_HMI_CRYO_TEMPERATURE_VOTE
{attribute 'TcHmiSymbol.Show'}
FUNCTION_BLOCK FB_METIS_HMI_CRYO_TEMPERATURE_VOTE
// VAR_INPUT
// 	{attribute 'TcHmiSymbol.Show'}
// 	in_all_temperature_names   : ARRAY [0..134] OF STRING;
// END_VAR
VAR_IN_OUT
	{attribute 'TcHmiSymbol.Show'}
	inout_sTemperatureStatRef : T_METIS_CRYO_TEMP_VOTE_STATUS;

END_VAR
VAR_IN_OUT CONSTANT
	inout_sCmdOver : FB_CRYO_CMD_OVERRIDE;
	inout_fbAlarmHandlerRef : FB_AlarmHandler;
END_VAR
VAR_OUTPUT
	{attribute 'TcHmiSymbol.ShowRecursively'}
	{attribute 'TcHmiSymbol.ReadOnly'}
	out_stat : T_HMI_METIS_TEMP_VOTER_STAT;
	
// 	{attribute 'TcHmiSymbol.ShowRecursively'}
// 	{attribute 'TcHmiSymbol.ReadOnly'}
// 	out_aTempIndexes:		ARRAY[0..4] OF INT;
// 	
// 	{attribute 'TcHmiSymbol.ShowRecursively'}
// 	{attribute 'TcHmiSymbol.ReadOnly'}
// 	out_nVoteMethod:		E_METIS_TEMP_VOTE_METHOD := E_METIS_TEMP_VOTE_METHOD.AVERAGE;
END_VAR
VAR	
	{attribute 'TcHmiSymbol.ShowRecursively'}
	ctrl : E_HMI_CRYO_SIMULATION_MODE_CTRL;;

	{attribute 'TcHmiSymbol.Show'}
	bChangeSimulatedTemperature : BOOL;
	{attribute 'TcHmiSymbol.Show'}
	lrSimulatedTemperatureInKelvinSetpoint : LREAL; // Requested simulated temperature

	{attribute 'TcHmiSymbol.Show'}
	{attribute 'TcHmiSymbol.ReadOnly'}
	sEventClassName : T_MaxString;

	{attribute 'TcHmiSymbol.Show'}
	{attribute 'TcHmiSymbol.ReadOnly'}
	sInstanceName : T_MaxString;

	{attribute 'TcHmiSymbol.Show'}
	bConfirmAllAlarms : BOOL;
	
	////////
	
	{attribute 'TcHmiSymbol.Show'}
	TestIndexes : ARRAY[0..4] OF E_ALL_METIS_TEMPERATURES;
	{attribute 'TcHmiSymbol.Show'} 
 	TestMethod : E_METIS_TEMP_VOTE_METHOD;


	
END_VAR



IF inout_sTemperatureStatRef.bReadConfig THEN
	
TestIndexes := inout_sTemperatureStatRef.aTempIndexes;
TestMethod  := inout_sTemperatureStatRef.nVoteMethod;
inout_sTemperatureStatRef.bReadConfig := FALSE;

ELSE

inout_sTemperatureStatRef.aTempIndexes := TestIndexes;
inout_sTemperatureStatRef.nVoteMethod  := TestMethod; 
END_IF

M_ProcessInput();

M_UpdateStatus();

sEventClassName := inout_fbAlarmHandlerRef.sEventClassName;
sInstanceName := inout_fbAlarmHandlerRef.sInstanceName;

IF bConfirmAllAlarms THEN
	bConfirmAllAlarms := FALSE;
	inout_fbAlarmHandlerRef.M_ConfirmAllAlarms();
END_IF

METHOD PRIVATE M_ProcessInput
{warning disable C0371}


IF ctrl = E_HMI_CRYO_SIMULATION_MODE_CTRL.NON_SIMULATED THEN
	inout_sCmdOver.M_SetAutoMode(TRUE);
	inout_sCmdOver.M_SetManualCmd(FALSE);
END_IF

IF ctrl = E_HMI_CRYO_SIMULATION_MODE_CTRL.SIMULATED THEN
	inout_sCmdOver.M_SetAutoMode(FALSE);
	inout_sCmdOver.M_SetManualCmd(TRUE);
END_IF

ctrl := E_HMI_CRYO_SIMULATION_MODE_CTRL.NONE;

IF bChangeSimulatedTemperature THEN
	inout_sTemperatureStatRef.lrSimTempK := lrSimulatedTemperatureInKelvinSetpoint;
	bChangeSimulatedTemperature := FALSE;
END_IF

{warning restore C0371}
END_METHOD

METHOD PRIVATE M_UpdateStatus
{warning disable C0371}

MEMCPY(destAddr := ADR(out_stat.temperature_stat),
	   srcAddr := ADR(inout_sTemperatureStatRef),
	   n := SIZEOF(inout_sTemperatureStatRef));

out_stat.cmd_over_stat.bEnable := inout_sCmdOver.out_bEnable;
out_stat.cmd_over_stat.bError := inout_sCmdOver.out_bError;
out_stat.cmd_over_stat.bInterlock := inout_sCmdOver.out_bInterlock;
out_stat.cmd_over_stat.bWarning := inout_sCmdOver.out_bWarning;
out_stat.cmd_over_stat.sMode := inout_sCmdOver.out_sMode;
out_stat.cmd_over_stat.sStatus := inout_sCmdOver.out_sStatus;
out_stat.cmd_over_stat.bPermitOn := inout_sCmdOver.bPermitOn;
out_stat.cmd_over_stat.bPermitOff := inout_sCmdOver.bPermitOff;
out_stat.cmd_over_stat.in_bEnable := inout_sCmdOver.in_bEnable;
out_stat.cmd_over_stat.bDisableBtnOn := inout_sCmdOver.bDisableBtnOn;
out_stat.cmd_over_stat.bDisableBtnOff := inout_sCmdOver.bDisableBtnOff;
out_stat.cmd_over_stat.bAutoMode := inout_sCmdOver.bAutoMode;
out_stat.cmd_over_stat.bEngMode := inout_sCmdOver.bEngMode;

{warning restore C0371}
END_METHOD

END_FUNCTION_BLOCK

// POUs/Devices/LakeShore_336/FB_METIS_LAKESHORES
FUNCTION_BLOCK FB_METIS_LAKESHORES
VAR_INPUT
END_VAR
VAR_OUTPUT
END_VAR
VAR
    ls_img_lm   : FB_METIS_LAKESHORE_336_TCP; // Lakeshore 336 of IMG LM detector
    ls_img_n    : FB_METIS_LAKESHORE_336_TCP; // Lakeshore 336 of IMG N detector
    ls_sca      : FB_METIS_LAKESHORE_336_TCP; // Lakeshore 336 of SCA detector
    
END_VAR

ls_img_lm(
    in_sName            := 'LS336_IMG_LM',
    in_nModel           := 336,
    in_nPeriod          := 1000,
    in_sCmdSuffix       := '$0A',
    in_sReplySuffix     := '$0A',
    in_sDeviceTcpIpAdr  := '172.16.0.111',
    in_nDeviceTcpPort   := 7777);
    
ls_img_n(
    in_sName            := 'LS336_IMG_N',
    in_nModel           := 336,
    in_nPeriod          := 1000,
    in_sCmdSuffix       := '$0A',
    in_sReplySuffix     := '$0A',
    in_sDeviceTcpIpAdr  := '172.16.0.112',
    in_nDeviceTcpPort   := 7777);

ls_sca(
    in_sName            := 'LS336_SCA',
    in_nModel           := 336,
    in_nPeriod          := 1000,
    in_sCmdSuffix       := '$0A',
    in_sReplySuffix     := '$0A',
    in_sDeviceTcpIpAdr  := '172.16.0.121',
    in_nDeviceTcpPort   := 7777);

END_FUNCTION_BLOCK

// POUs/Devices/LakeShore_336/FB_METIS_LAKESHORE_336_TCP
FUNCTION_BLOCK FB_METIS_LAKESHORE_336_TCP EXTENDS FB_LAKESHORE_BASE
VAR_INPUT
	{attribute 'OPC.UA.DA' := '0'}
	in_sDeviceTcpIpAdr: STRING(16);		// Lakeshore IP address, e.g. '192.168.0.80'
	{attribute 'OPC.UA.DA' := '0'}
    in_nDeviceTcpPort:	UINT;			// Lakeshore Tcp port, default 7777 
END_VAR
VAR_OUTPUT
END_VAR
VAR
	{attribute 'OPC.UA.DA' := '0'}
	comm:		FB_TCP_CLIENT;			// Instance of Tcp comm FB. OPC UA Disabled!!!
	
	// Temperature outputs so that Temp specific FBs can read and validate the temperature readings
	Temp_A 		AT%Q*:	LREAL;
	Temp_B 		AT%Q*:	LREAL;
	Temp_C 		AT%Q*:	LREAL;
	Temp_D 		AT%Q*:	LREAL;
    
    // toggle outputs
    q_bValid_A AT%Q*    : BOOL;
    q_bValid_B AT%Q*    : BOOL;
    q_bValid_C AT%Q*    : BOOL;
    q_bValid_D AT%Q*    : BOOL;
    
    // extra diagnostics
    nCommPreviouStatus : E_RS_COMM_STATUS;
    nCommErrors : LINT := 0;

END_VAR


(* Execute comm instance *)
comm(	in_bSimulation		:= in_bSimulation,
		in_sDeviceTcpIpAdr	:= in_sDeviceTcpIpAdr,
		in_nDeviceTcpPort	:= in_nDeviceTcpPort, 
		in_sCmdSuffix		:= in_sCmdSuffix, 
		in_sReplySuffix		:= in_sReplySuffix,
		in_nPollingDelay 	:= 10,
		in_nTimeout			:= 2000);
		



// Execute the base class object FB_RS_BASE
SUPER^();

M_SetTemperatureOutputs();

IF comm.stat.nStatus = E_RS_COMM_STATUS.ERROR AND nCommPreviouStatus <> E_RS_COMM_STATUS.ERROR THEN
    nCommErrors := nCommErrors + 1;
END_IF
nCommPreviouStatus := comm.stat.nStatus;

METHOD M_Configure
VAR_INPUT
END_VAR
VAR
	// This is OK for models 224 and 336
	cmdList_Init_224:	ARRAY [1..8] OF T_LAKESHORE_COMMAND := [
							(cmd := 'MODE 1', 	nReplies := 0, 	nValues := 0,	offset := 0),
							(cmd := '*IDN?', 	nReplies := 1, 	nValues := 1,	offset := 0),
							(cmd := '', 		nReplies := 0, 	nValues := 0,	offset := 0),
							(cmd := '', 		nReplies := 0, 	nValues := 0,	offset := 0),
							(cmd := '', 		nReplies := 0, 	nValues := 0,	offset := 0),
							(cmd := '', 		nReplies := 0, 	nValues := 0,	offset := 0),
							(cmd := '', 		nReplies := 0, 	nValues := 0,	offset := 0),
							(cmd := '', 		nReplies := 0, 	nValues := 0,	offset := 0)];

	cmdList_Init_336:	ARRAY [1..8] OF T_LAKESHORE_COMMAND := [
							(cmd := 'MODE 1', 	nReplies := 0, 	nValues := 0,	offset := 0),
							(cmd := '*IDN?', 	nReplies := 1, 	nValues := 1,	offset := 0),
							(cmd := '', 		nReplies := 0, 	nValues := 0,	offset := 0),
							(cmd := '', 		nReplies := 0, 	nValues := 0,	offset := 0),
							(cmd := '', 		nReplies := 0, 	nValues := 0,	offset := 0),
							(cmd := '', 		nReplies := 0, 	nValues := 0,	offset := 0),
							(cmd := '', 		nReplies := 0, 	nValues := 0,	offset := 0),
							(cmd := '', 		nReplies := 0, 	nValues := 0,	offset := 0)];


	(*	List of READ commands *)
	(* Lakeshore 218 commands:
		Command "KRDG? 0" requests all 8 temperature values in K.
		Command "CRDG? 0" requests all 8 temperature values in C.
		Reply format: 
			+nn.nnn,+nn.nnn,+nn.nnn,+nn.nnn,+nn.nnn,+nn.nnn,+nn.nnn,+nn.nnn<CR><LF>
	*)

	cmdList_Read_224:	ARRAY [1..16] OF T_LAKESHORE_COMMAND := [
							(cmd := 'KRDG? 0', 	nReplies := 1, 	nValues := 12,	offset := 0),
							(cmd := 'CRDG? 0', 	nReplies := 1, 	nValues := 12,	offset := 12),
							(cmd := '', 		nReplies := 0, 	nValues := 0,	offset := 0),
							(cmd := '', 		nReplies := 0, 	nValues := 0,	offset := 0),
							(cmd := '', 		nReplies := 0, 	nValues := 0,	offset := 0),
							(cmd := '', 		nReplies := 0, 	nValues := 0,	offset := 0),
							(cmd := '', 		nReplies := 0, 	nValues := 0,	offset := 0),
							(cmd := '', 		nReplies := 0, 	nValues := 0,	offset := 0),
							(cmd := '', 		nReplies := 0, 	nValues := 0,	offset := 0),
							(cmd := '', 		nReplies := 0, 	nValues := 0,	offset := 0),
							(cmd := '', 		nReplies := 0, 	nValues := 0,	offset := 0),
							(cmd := '', 		nReplies := 0, 	nValues := 0,	offset := 0),
							(cmd := '', 		nReplies := 0, 	nValues := 0,	offset := 0),
							(cmd := '', 		nReplies := 0, 	nValues := 0,	offset := 0),
							(cmd := '', 		nReplies := 0, 	nValues := 0,	offset := 0),
							(cmd := '', 		nReplies := 0, 	nValues := 0,	offset := 0)];

	cmdList_Read_336:	ARRAY [1..16] OF T_LAKESHORE_COMMAND := [
							(cmd := 'KRDG? A', 	nReplies := 1, 	nValues := 1,	offset := 0),
							(cmd := 'KRDG? B', 	nReplies := 1, 	nValues := 1,	offset := 1),
							(cmd := 'SETP? 1', 	nReplies := 1, 	nValues := 1,	offset := 2),
							(cmd := 'PID? 1', 	nReplies := 1, 	nValues := 3,	offset := 3),
							(cmd := 'RAMP? 1', 	nReplies := 1, 	nValues := 2,	offset := 6),
							(cmd := 'RANGE? 1', nReplies := 1, 	nValues := 1,	offset := 8),
							(cmd := 'HTR? 1', 	nReplies := 1, 	nValues := 1,	offset := 9),
							(cmd := 'SETP? 2', 	nReplies := 1, 	nValues := 1,	offset := 10),
							(cmd := 'PID? 2', 	nReplies := 1, 	nValues := 3,	offset := 11),
							(cmd := 'RAMP? 2', 	nReplies := 1, 	nValues := 2,	offset := 14),
							(cmd := 'RANGE? 2', nReplies := 1, 	nValues := 1,	offset := 16),
							(cmd := 'HTR? 2', 	nReplies := 1, 	nValues := 1,	offset := 17),
							(cmd := 'AOUT? 3', 	nReplies := 1, 	nValues := 1,	offset := 18),
							(cmd := 'AOUT? 4', 	nReplies := 1, 	nValues := 1,	offset := 19),
							(cmd := 'KRDG? C',  nReplies := 1,  nValues := 1,   offset := 20),
                            (cmd := 'KRDG? D',  nReplies := 1,  nValues := 1,   offset := 21)];

	
END_VAR
// Execute base FB M_Configure().
// This will set cfg.nModel, etc.
SUPER^.M_Configure();

// TODO
// Populate cfg.cmdList_Init and cmdList_Read tables for the specific cfg.nModel.
IF cfg.nModel = 224 THEN
	cfg.cmdList_Init	:= cmdList_Init_224;
	cfg.cmdList_Read	:= cmdList_Read_224;
ELSIF cfg.nModel = 336 THEN
	cfg.cmdList_Init	:= cmdList_Init_336;
	cfg.cmdList_Read	:= cmdList_Read_336;
END_IF


// Set pointers to comm, i.e.
ptrCommCfg	:= ADR(comm.cfg);	(* Pointer to comm.cfg instance *)
ptrCommCtrl	:= ADR(comm.ctrl);	(* Pointer to comm.ctrl instance *)
ptrCommStat	:= ADR(comm.stat);	(* Pointer to comm.stat instance *)

// Set comm suffixes for commands and replies
ptrCommCfg^.sCmdSuffix		:= in_sCmdSuffix;
ptrCommCfg^.sReplySuffix	:= in_sReplySuffix;
END_METHOD

METHOD M_GetCommInitialised : BOOL
VAR_INPUT
END_VAR
M_GetCommInitialised	:= comm.M_GetInitialised();
END_METHOD

METHOD M_GetCommStatus : E_RS_COMM_STATUS
VAR_INPUT
END_VAR
M_GetCommStatus	:= comm.M_GetStatus();
END_METHOD

METHOD M_SetTemperatureOutputs
VAR_INPUT
END_VAR
Temp_A := stat.lrArrReadings[0].lrValue;
Temp_B := stat.lrArrReadings[1].lrValue;
Temp_C := stat.lrArrReadings[20].lrValue;
Temp_D := stat.lrArrReadings[21].lrValue;

q_bValid_A := stat.bActive 
                AND comm.stat.nStatus <> E_RS_COMM_STATUS.ERROR 
                AND (    stat.nSubstate = E_RS_BASE_SUBSTATE.OP_MONITORING 
                     OR  stat.nSubstate = E_RS_BASE_SUBSTATE.OP_MONITORING_USER);
q_bValid_B := q_bValid_A;  // no distinction possible
q_bValid_C := q_bValid_A;  // no distinction possible
q_bValid_D := q_bValid_A;  // no distinction possible
END_METHOD

METHOD M_UpdateStatus
VAR_INPUT
END_VAR
// TODO
//
// Copy values from stat.lrReadings to correspondig stat variables.
// Check M_Configure(). It has to match!
//
// This is an example for model 340.
// This method has to match the list of commands in T_LAKESHORE_CFG::cmdList_Read
IF cfg.nModel = 224 THEN
	// Nothing to do.
	// NOTE: 12 readings [K]: stat.lrArrReadings[0..11].lrValue
	// NOTE: 12 readings [C]: stat.lrArrReadings[12..23].lrValue
	;	
ELSIF cfg.nModel = 336 THEN
	// TODO NOTE: Only loop 1 is handled !!!
	stat.lrKRDG_A		:= stat.lrArrReadings[0].lrValue;
	stat.lrCRDG_A		:= stat.lrKRDG_A - 273.15;
	stat.lrKRDG_B		:= stat.lrArrReadings[1].lrValue;
	stat.lrCRDG_B		:= stat.lrKRDG_B - 273.15;
	// Loop 1
	stat.lrSETP			:= stat.lrArrReadings[2].lrValue;
	stat.nPID_P			:= LREAL_TO_UINT(stat.lrArrReadings[3].lrValue);
	stat.nPID_I			:= LREAL_TO_UINT(stat.lrArrReadings[4].lrValue);
	stat.nPID_D			:= LREAL_TO_UINT(stat.lrArrReadings[5].lrValue);
	stat.bRAMP_On		:= LREAL_TO_BOOL(stat.lrArrReadings[6].lrValue);
	stat.lrRAMP_Rate	:= stat.lrArrReadings[7].lrValue;
	stat.nRANGE			:= LREAL_TO_UINT(stat.lrArrReadings[8].lrValue);
	stat.lrHTR			:= stat.lrArrReadings[9].lrValue;
	// Loop 2
	stat.lrSETP2		:= stat.lrArrReadings[10].lrValue;
	stat.nPID2_P		:= LREAL_TO_UINT(stat.lrArrReadings[11].lrValue);
	stat.nPID2_I		:= LREAL_TO_UINT(stat.lrArrReadings[12].lrValue);
	stat.nPID2_D		:= LREAL_TO_UINT(stat.lrArrReadings[13].lrValue);
	stat.bRAMP2_On		:= LREAL_TO_BOOL(stat.lrArrReadings[14].lrValue);
	stat.lrRAMP2_Rate	:= stat.lrArrReadings[15].lrValue;
	stat.nRANGE2		:= LREAL_TO_UINT(stat.lrArrReadings[16].lrValue);
	stat.lrHTR2			:= stat.lrArrReadings[17].lrValue;
	// Outputs
	stat.lrAOUT3		:= stat.lrArrReadings[18].lrValue;
	stat.lrAOUT4		:= stat.lrArrReadings[19].lrValue;

END_IF
END_METHOD

END_FUNCTION_BLOCK

